LIN {X 0,Y 315.719,Z 733.66,A -85,B 0,C 180,E1 14074.745,E2 14074.745} C_VEL
LIN {X 0,Y 317.887,Z 739.054,A -85,B 0,C 180,E1 14075.526,E2 14075.526} C_VEL
LIN {X 0,Y 320.748,Z 743.078,A -85,B 0,C 180,E1 14076.392,E2 14076.392} C_VEL
LIN {X 0,Y 337.492,Z 768.828,A -85,B 0,C 180,E1 14081.01,E2 14081.01} C_VEL
LIN {X 0,Y 351.27,Z 797.337,A -85,B 0,C 180,E1 14085.073,E2 14085.073} C_VEL
LIN {X 0,Y 359.237,Z 823.028,A -85,B 0,C 180,E1 14088.326,E2 14088.326} C_VEL
LIN {X 0,Y 352.116,Z 857.888,A -85,B 0,C 180,E1 14091.071,E2 14091.071} C_VEL
LIN {X 0,Y 344.17,Z 888.383,A -85,B 0,C 180,E1 14094.581,E2 14094.581} C_VEL
LIN {X 0,Y 336.227,Z 914.82,A -85,B 0,C 180,E1 14098.833,E2 14098.833} C_VEL
LIN {X 0,Y 328.748,Z 938.426,A -85,B 0,C 180,E1 14104.142,E2 14104.142} C_VEL
LIN {X 0,Y 323.256,Z 956.658,A -85,B 0,C 180,E1 14110.032,E2 14110.032} C_VEL
LIN {X 0,Y 319.91,Z 969.689,A -85,B 0,C 180,E1 14116.312,E2 14116.312} C_VEL
LIN {X 0,Y 318.308,Z 977.967,A -85,B 0,C 180,E1 14123.171,E2 14123.171} C_VEL
LIN {X 0,Y 318.122,Z 980.655,A -85,B 0,C 180,E1 14130,E2 14130} C_VEL
LIN {X 0,Y 318.325,Z 977.878,A -85,B 0,C 180,E1 14136.83,E2 14136.83} C_VEL
LIN {X 0,Y 319.962,Z 969.528,A -85,B 0,C 180,E1 14143.687,E2 14143.687} C_VEL
LIN {X 0,Y 323.345,Z 956.356,A -85,B 0,C 180,E1 14149.986,E2 14149.986} C_VEL
LIN {X 0,Y 328.917,Z 937.87,A -85,B 0,C 180,E1 14155.897,E2 14155.897} C_VEL
LIN {X 0,Y 336.458,Z 913.934,A -85,B 0,C 180,E1 14161.232,E2 14161.232} C_VEL
LIN {X 0,Y 344.929,Z 885.442,A -85,B 0,C 180,E1 14165.728,E2 14165.728} C_VEL
LIN {X 0,Y 353.166,Z 852.828,A -85,B 0,C 180,E1 14169.299,E2 14169.299} C_VEL
LIN {X 0,Y 359.003,Z 821.032,A -85,B 0,C 180,E1 14171.77,E2 14171.77} C_VEL
LIN {X 0,Y 348.714,Z 791.49,A -85,B 0,C 180,E1 14175.622,E2 14175.622} C_VEL
LIN {X 0,Y 333.855,Z 762.92,A -85,B 0,C 180,E1 14179.841,E2 14179.841} C_VEL
LIN {X 0,Y 318.479,Z 739.646,A -85,B 0,C 180,E1 14184.163,E2 14184.163} C_VEL
LIN {X 0,Y 315.762,Z 734.408,A -85,B 0,C 180,E1 14185.064,E2 14185.064} C_VEL
LIN {X 0,Y 315.891,Z 733.66,A -85,B 0,C 180,E1 14191.354,E2 14191.354} C_VEL
LIN {X 0,Y 316.196,Z 733.66,A -85,B 0,C 180,E1 14197.47,E2 14197.47} C_VEL
LIN {X 0,Y 316.495,Z 733.66,A -85,B 0,C 180,E1 14203.314,E2 14203.314} C_VEL
LIN {X 0,Y 317.022,Z 733.66,A -85,B 0,C 180,E1 14211.757,E2 14211.757} C_VEL
LIN {X 0,Y 317.696,Z 733.66,A -85,B 0,C 180,E1 14219.994,E2 14219.994} C_VEL
LIN {X 0,Y 317.039,Z 733.66,A -85,B 0,C 180,E1 14228.231,E2 14228.231} C_VEL
LIN {X 0,Y 316.543,Z 733.66,A -85,B 0,C 180,E1 14236.671,E2 14236.671} C_VEL
LIN {X 0,Y 316.1,Z 733.66,A -85,B 0,C 180,E1 14244.482,E2 14244.482} C_VEL
LIN {X 0,Y 315.775,Z 733.66,A -85,B 0,C 180,E1 14251.823,E2 14251.823} C_VEL
LIN {X 0,Y 315.754,Z 733.66,A -85,B 0,C 180,E1 14254.342,E2 14254.342} C_VEL
LIN {X 0,Y 317.927,Z 739.136,A -85,B 0,C 180,E1 14255.152,E2 14255.152} C_VEL
LIN {X 0,Y 321.023,Z 743.491,A -85,B 0,C 180,E1 14256.083,E2 14256.083} C_VEL
LIN {X 0,Y 336.553,Z 767.239,A -85,B 0,C 180,E1 14260.305,E2 14260.305} C_VEL
LIN {X 0,Y 350.017,Z 791.741,A -85,B 0,C 180,E1 14263.573,E2 14263.573} C_VEL
LIN {X 0,Y 360.355,Z 827.54,A -85,B 0,C 180,E1 14267.003,E2 14267.003} C_VEL
LIN {X 0,Y 354.186,Z 864.729,A -85,B 0,C 180,E1 14269.179,E2 14269.179} C_VEL
LIN {X 0,Y 346.202,Z 898.964,A -85,B 0,C 180,E1 14272.245,E2 14272.245} C_VEL
LIN {X 0,Y 337.789,Z 929.303,A -85,B 0,C 180,E1 14276.16,E2 14276.16} C_VEL
LIN {X 0,Y 329.891,Z 956.501,A -85,B 0,C 180,E1 14281.15,E2 14281.15} C_VEL
LIN {X 0,Y 323.714,Z 978.764,A -85,B 0,C 180,E1 14286.938,E2 14286.938} C_VEL
LIN {X 0,Y 319.815,Z 996.193,A -85,B 0,C 180,E1 14293.497,E2 14293.497} C_VEL
LIN {X 0,Y 318.446,Z 1005.836,A -85,B 0,C 180,E1 14299.036,E2 14299.036} C_VEL
LIN {X 0,Y 318.166,Z 1011.498,A -85,B 0,C 180,E1 14304.538,E2 14304.538} C_VEL
LIN {X 0,Y 318.196,Z 1013.428,A -85,B 0,C 180,E1 14310,E2 14310} C_VEL
LIN {X 0,Y 318.188,Z 1011.507,A -85,B 0,C 180,E1 14315.461,E2 14315.461} C_VEL
LIN {X 0,Y 318.486,Z 1005.851,A -85,B 0,C 180,E1 14320.962,E2 14320.962} C_VEL
LIN {X 0,Y 320.15,Z 994.65,A -85,B 0,C 180,E1 14327.192,E2 14327.192} C_VEL
LIN {X 0,Y 324.095,Z 977.701,A -85,B 0,C 180,E1 14333.397,E2 14333.397} C_VEL
LIN {X 0,Y 330.329,Z 955.266,A -85,B 0,C 180,E1 14339.134,E2 14339.134} C_VEL
LIN {X 0,Y 338.372,Z 927.731,A -85,B 0,C 180,E1 14344.078,E2 14344.078} C_VEL
LIN {X 0,Y 344.691,Z 905.27,A -85,B 0,C 180,E1 14347.058,E2 14347.058} C_VEL
LIN {X 0,Y 345.028,Z 891.788,A -85,B 0,C 180,E1 14348.915,E2 14348.915} C_VEL
LIN {X 0,Y 344.878,Z 879.547,A -85,B 0,C 180,E1 14350.45,E2 14350.45} C_VEL
LIN {X 0,Y 345.262,Z 877.652,A -85,B 0,C 180,E1 14350.624,E2 14350.624} C_VEL
LIN {X 0,Y 352.782,Z 841.115,A -85,B 0,C 180,E1 14353.157,E2 14353.157} C_VEL
LIN {X 0,Y 354.632,Z 826.28,A -85,B 0,C 180,E1 14353.945,E2 14353.945} C_VEL
LIN {X 0,Y 353.828,Z 815.884,A -85,B 0,C 180,E1 14354.939,E2 14354.939} C_VEL
LIN {X 0,Y 354.413,Z 805.731,A -85,B 0,C 180,E1 14356.89,E2 14356.89} C_VEL
LIN {X 0,Y 352.564,Z 801.602,A -85,B 0,C 180,E1 14359.906,E2 14359.906} C_VEL
LIN {X 0,Y 352.295,Z 802.737,A -85,B 0,C 180,E1 14363.018,E2 14363.018} C_VEL
LIN {X 0,Y 352.883,Z 809.058,A -85,B 0,C 180,E1 14365.545,E2 14365.545} C_VEL
LIN {X 0,Y 343.129,Z 843.636,A -85,B 0,C 180,E1 14368.963,E2 14368.963} C_VEL
LIN {X 0,Y 335.37,Z 867.34,A -85,B 0,C 180,E1 14372.482,E2 14372.482} C_VEL
LIN {X 0,Y 327.758,Z 887.089,A -85,B 0,C 180,E1 14376.888,E2 14376.888} C_VEL
LIN {X 0,Y 321.86,Z 900.268,A -85,B 0,C 180,E1 14381.494,E2 14381.494} C_VEL
LIN {X 0,Y 317.622,Z 908.248,A -85,B 0,C 180,E1 14386.218,E2 14386.218} C_VEL
LIN {X 0,Y 314.61,Z 911.796,A -85,B 0,C 180,E1 14391.705,E2 14391.705} C_VEL
LIN {X 0,Y 313.23,Z 909.746,A -85,B 0,C 180,E1 14397.236,E2 14397.236} C_VEL
LIN {X 0,Y 313.169,Z 901.828,A -85,B 0,C 180,E1 14402.777,E2 14402.777} C_VEL
LIN {X 0,Y 314.276,Z 888.435,A -85,B 0,C 180,E1 14407.967,E2 14407.967} C_VEL
LIN {X 0,Y 316.237,Z 870.789,A -85,B 0,C 180,E1 14412.448,E2 14412.448} C_VEL
LIN {X 0,Y 319.015,Z 847.121,A -85,B 0,C 180,E1 14416.55,E2 14416.55} C_VEL
LIN {X 0,Y 321.875,Z 820.749,A -85,B 0,C 180,E1 14419.65,E2 14419.65} C_VEL
LIN {X 0,Y 324.187,Z 789.991,A -85,B 0,C 180,E1 14421.945,E2 14421.945} C_VEL
LIN {X 0,Y 310.002,Z 740.414,A -85,B 0,C 180,E1 14425.18,E2 14425.18} C_VEL
LIN {X 0,Y 308.125,Z 733.66,A -85,B 0,C 180,E1 14425.647,E2 14425.647} C_VEL
LIN {X 0,Y 307.834,Z 733.76,A -85,B 0,C 180,E1 14432.566,E2 14432.566} C_VEL
LIN {X 0,Y 310.075,Z 739.153,A -85,B 0,C 180,E1 14433.438,E2 14433.438} C_VEL
LIN {X 0,Y 312.739,Z 742.517,A -85,B 0,C 180,E1 14434.311,E2 14434.311} C_VEL
LIN {X 0,Y 328.649,Z 766.861,A -85,B 0,C 180,E1 14439.098,E2 14439.098} C_VEL
LIN {X 0,Y 342.598,Z 793.742,A -85,B 0,C 180,E1 14443.318,E2 14443.318} C_VEL
LIN {X 0,Y 352.285,Z 821.897,A -85,B 0,C 180,E1 14447.171,E2 14447.171} C_VEL
LIN {X 0,Y 352.391,Z 828.572,A -85,B 0,C 180,E1 14447.809,E2 14447.809} C_VEL
LIN {X 0,Y 344.891,Z 862.553,A -85,B 0,C 180,E1 14450.676,E2 14450.676} C_VEL
LIN {X 0,Y 336.417,Z 893.037,A -85,B 0,C 180,E1 14454.39,E2 14454.39} C_VEL
LIN {X 0,Y 327.713,Z 920.477,A -85,B 0,C 180,E1 14459.161,E2 14459.161} C_VEL
LIN {X 0,Y 320.127,Z 943.273,A -85,B 0,C 180,E1 14464.807,E2 14464.807} C_VEL
LIN {X 0,Y 314.687,Z 960.699,A -85,B 0,C 180,E1 14471.049,E2 14471.049} C_VEL
LIN {X 0,Y 311.683,Z 972.269,A -85,B 0,C 180,E1 14477.374,E2 14477.374} C_VEL
LIN {X 0,Y 310.313,Z 979.325,A -85,B 0,C 180,E1 14484.4,E2 14484.4} C_VEL
LIN {X 0,Y 310.245,Z 981.06,A -85,B 0,C 180,E1 14490,E2 14490} C_VEL
LIN {X 0,Y 310.473,Z 978.285,A -85,B 0,C 180,E1 14497.003,E2 14497.003} C_VEL
LIN {X 0,Y 312.248,Z 969.827,A -85,B 0,C 180,E1 14504.104,E2 14504.104} C_VEL
LIN {X 0,Y 316.145,Z 955.711,A -85,B 0,C 180,E1 14510.9,E2 14510.9} C_VEL
LIN {X 0,Y 322.48,Z 935.952,A -85,B 0,C 180,E1 14517.134,E2 14517.134} C_VEL
LIN {X 0,Y 330.754,Z 911.07,A -85,B 0,C 180,E1 14522.574,E2 14522.574} C_VEL
LIN {X 0,Y 339.489,Z 882.48,A -85,B 0,C 180,E1 14526.939,E2 14526.939} C_VEL
LIN {X 0,Y 347.64,Z 850.852,A -85,B 0,C 180,E1 14530.339,E2 14530.339} C_VEL
LIN {X 0,Y 352.866,Z 824.113,A -85,B 0,C 180,E1 14532.427,E2 14532.427} C_VEL
LIN {X 0,Y 342.854,Z 794.622,A -85,B 0,C 180,E1 14536.463,E2 14536.463} C_VEL
LIN {X 0,Y 328.84,Z 767.242,A -85,B 0,C 180,E1 14540.716,E2 14540.716} C_VEL
LIN {X 0,Y 314.245,Z 745.05,A -85,B 0,C 180,E1 14545.044,E2 14545.044} C_VEL
LIN {X 0,Y 310.585,Z 739.636,A -85,B 0,C 180,E1 14546.254,E2 14546.254} C_VEL
LIN {X 0,Y 307.873,Z 734.455,A -85,B 0,C 180,E1 14547.245,E2 14547.245} C_VEL
LIN {X 0,Y 308.049,Z 733.66,A -85,B 0,C 180,E1 14553.74,E2 14553.74} C_VEL
LIN {X 0,Y 308.391,Z 733.66,A -85,B 0,C 180,E1 14559.893,E2 14559.893} C_VEL
LIN {X 0,Y 308.644,Z 733.66,A -85,B 0,C 180,E1 14565.796,E2 14565.796} C_VEL
LIN {X 0,Y 309.312,Z 733.66,A -85,B 0,C 180,E1 14574.376,E2 14574.376} C_VEL
LIN {X 0,Y 309.792,Z 733.66,A -85,B 0,C 180,E1 14579.994,E2 14579.994} C_VEL
LIN {X 0,Y 309.097,Z 733.66,A -85,B 0,C 180,E1 14588.444,E2 14588.444} C_VEL
LIN {X 0,Y 308.596,Z 733.66,A -85,B 0,C 180,E1 14597.113,E2 14597.113} C_VEL
LIN {X 0,Y 308.217,Z 733.66,A -85,B 0,C 180,E1 14603.133,E2 14603.133} C_VEL
LIN {X 0,Y 307.864,Z 733.66,A -85,B 0,C 180,E1 14611.215,E2 14611.215} C_VEL
LIN {X 0,Y 307.871,Z 733.66,A -85,B 0,C 180,E1 14612.165,E2 14612.165} C_VEL
LIN {X 0,Y 310.1,Z 739.211,A -85,B 0,C 180,E1 14613.067,E2 14613.067} C_VEL
LIN {X 0,Y 312.757,Z 742.554,A -85,B 0,C 180,E1 14613.934,E2 14613.934} C_VEL
LIN {X 0,Y 329.952,Z 768.564,A -85,B 0,C 180,E1 14618.991,E2 14618.991} C_VEL
LIN {X 0,Y 344.988,Z 795.969,A -85,B 0,C 180,E1 14622.854,E2 14622.854} C_VEL
LIN {X 0,Y 354.429,Z 830.867,A -85,B 0,C 180,E1 14626.343,E2 14626.343} C_VEL
LIN {X 0,Y 347.762,Z 866.235,A -85,B 0,C 180,E1 14628.466,E2 14628.466} C_VEL
LIN {X 0,Y 339.854,Z 898.559,A -85,B 0,C 180,E1 14631.411,E2 14631.411} C_VEL
LIN {X 0,Y 331.048,Z 929.012,A -85,B 0,C 180,E1 14635.397,E2 14635.397} C_VEL
LIN {X 0,Y 322.614,Z 956.671,A -85,B 0,C 180,E1 14640.588,E2 14640.588} C_VEL
LIN {X 0,Y 316.476,Z 977.674,A -85,B 0,C 180,E1 14646.151,E2 14646.151} C_VEL
LIN {X 0,Y 312.377,Z 994.208,A -85,B 0,C 180,E1 14652.365,E2 14652.365} C_VEL
LIN {X 0,Y 310.585,Z 1005.423,A -85,B 0,C 180,E1 14658.755,E2 14658.755} C_VEL
LIN {X 0,Y 310.267,Z 1011.089,A -85,B 0,C 180,E1 14664.399,E2 14664.399} C_VEL
LIN {X 0,Y 310.314,Z 1013.022,A -85,B 0,C 180,E1 14670,E2 14670} C_VEL
LIN {X 0,Y 310.288,Z 1011.099,A -85,B 0,C 180,E1 14675.6,E2 14675.6} C_VEL
LIN {X 0,Y 310.832,Z 1004.069,A -85,B 0,C 180,E1 14682.218,E2 14682.218} C_VEL
LIN {X 0,Y 313.101,Z 991.048,A -85,B 0,C 180,E1 14689.051,E2 14689.051} C_VEL
LIN {X 0,Y 317.903,Z 972.612,A -85,B 0,C 180,E1 14695.381,E2 14695.381} C_VEL
LIN {X 0,Y 324.742,Z 949.962,A -85,B 0,C 180,E1 14700.855,E2 14700.855} C_VEL
LIN {X 0,Y 333.393,Z 921.91,A -85,B 0,C 180,E1 14705.671,E2 14705.671} C_VEL
LIN {X 0,Y 342.039,Z 890.249,A -85,B 0,C 180,E1 14709.475,E2 14709.475} C_VEL
LIN {X 0,Y 345.262,Z 877.652,A -85,B 0,C 180,E1 14710.624,E2 14710.624} C_VEL
LIN {X 0,Y 345.636,Z 862.952,A -85,B 0,C 180,E1 14712.213,E2 14712.213} C_VEL
LIN {X 0,Y 345.686,Z 847.734,A -85,B 0,C 180,E1 14713.652,E2 14713.652} C_VEL
LIN {X 0,Y 348.589,Z 827.915,A -85,B 0,C 180,E1 14714.778,E2 14714.778} C_VEL
LIN {X 0,Y 349.864,Z 816.657,A -85,B 0,C 180,E1 14716.342,E2 14716.342} C_VEL
LIN {X 0,Y 350.407,Z 812.2,A -85,B 0,C 180,E1 14717.27,E2 14717.27} C_VEL
LIN {X 0,Y 349.152,Z 809.136,A -85,B 0,C 180,E1 14719.433,E2 14719.433} C_VEL
LIN {X 0,Y 348.638,Z 809.515,A -85,B 0,C 180,E1 14722.564,E2 14722.564} C_VEL
LIN {X 0,Y 348.845,Z 813.277,A -85,B 0,C 180,E1 14724.507,E2 14724.507} C_VEL
LIN {X 0,Y 336.466,Z 851.174,A -85,B 0,C 180,E1 14728.657,E2 14728.657} C_VEL
LIN {X 0,Y 327.878,Z 874.081,A -85,B 0,C 180,E1 14732.506,E2 14732.506} C_VEL
LIN {X 0,Y 319.961,Z 892.066,A -85,B 0,C 180,E1 14737.029,E2 14737.029} C_VEL
LIN {X 0,Y 313.274,Z 905.19,A -85,B 0,C 180,E1 14742.426,E2 14742.426} C_VEL
LIN {X 0,Y 309.131,Z 911.475,A -85,B 0,C 180,E1 14747.274,E2 14747.274} C_VEL
LIN {X 0,Y 306.931,Z 913.336,A -85,B 0,C 180,E1 14751.496,E2 14751.496} C_VEL
LIN {X 0,Y 305.425,Z 910.977,A -85,B 0,C 180,E1 14757.165,E2 14757.165} C_VEL
LIN {X 0,Y 305.353,Z 902.819,A -85,B 0,C 180,E1 14762.848,E2 14762.848} C_VEL
LIN {X 0,Y 306.49,Z 889.121,A -85,B 0,C 180,E1 14768.171,E2 14768.171} C_VEL
LIN {X 0,Y 308.771,Z 869.532,A -85,B 0,C 180,E1 14773.114,E2 14773.114} C_VEL
LIN {X 0,Y 311.579,Z 846.035,A -85,B 0,C 180,E1 14777.139,E2 14777.139} C_VEL
LIN {X 0,Y 314.582,Z 818.438,A -85,B 0,C 180,E1 14780.308,E2 14780.308} C_VEL
LIN {X 0,Y 316.404,Z 789.468,A -85,B 0,C 180,E1 14782.459,E2 14782.459} C_VEL
LIN {X 0,Y 300.116,Z 733.66,A -85,B 0,C 180,E1 14786.454,E2 14786.454} C_VEL
LIN {X 0,Y 299.966,Z 733.66,A -85,B 0,C 180,E1 14790.097,E2 14790.097} C_VEL
LIN {X 0,Y 301.982,Z 738.935,A -85,B 0,C 180,E1 14791.005,E2 14791.005} C_VEL
LIN {X 0,Y 305.006,Z 742.493,A -85,B 0,C 180,E1 14792.101,E2 14792.101} C_VEL
LIN {X 0,Y 320.547,Z 765.584,A -85,B 0,C 180,E1 14797.201,E2 14797.201} C_VEL
LIN {X 0,Y 334.503,Z 791.877,A -85,B 0,C 180,E1 14801.673,E2 14801.673} C_VEL
LIN {X 0,Y 344.06,Z 817.214,A -85,B 0,C 180,E1 14805.397,E2 14805.397} C_VEL
LIN {X 0,Y 346.837,Z 827.807,A -85,B 0,C 180,E1 14806.856,E2 14806.856} C_VEL
LIN {X 0,Y 338.826,Z 862.802,A -85,B 0,C 180,E1 14809.812,E2 14809.812} C_VEL
LIN {X 0,Y 330.004,Z 893.431,A -85,B 0,C 180,E1 14813.589,E2 14813.589} C_VEL
LIN {X 0,Y 320.835,Z 920.937,A -85,B 0,C 180,E1 14818.439,E2 14818.439} C_VEL
LIN {X 0,Y 312.87,Z 943.681,A -85,B 0,C 180,E1 14824.181,E2 14824.181} C_VEL
LIN {X 0,Y 307.124,Z 961.108,A -85,B 0,C 180,E1 14830.564,E2 14830.564} C_VEL
LIN {X 0,Y 303.876,Z 972.875,A -85,B 0,C 180,E1 14837.201,E2 14837.201} C_VEL
LIN {X 0,Y 302.441,Z 979.732,A -85,B 0,C 180,E1 14844.254,E2 14844.254} C_VEL
LIN {X 0,Y 302.37,Z 981.466,A -85,B 0,C 180,E1 14850,E2 14850} C_VEL
LIN {X 0,Y 302.609,Z 978.694,A -85,B 0,C 180,E1 14857.186,E2 14857.186} C_VEL
LIN {X 0,Y 304.494,Z 970.35,A -85,B 0,C 180,E1 14864.397,E2 14864.397} C_VEL
LIN {X 0,Y 308.649,Z 956.253,A -85,B 0,C 180,E1 14871.381,E2 14871.381} C_VEL
LIN {X 0,Y 315.139,Z 937.036,A -85,B 0,C 180,E1 14877.617,E2 14877.617} C_VEL
LIN {X 0,Y 323.286,Z 913.635,A -85,B 0,C 180,E1 14882.919,E2 14882.919} C_VEL
LIN {X 0,Y 332.374,Z 885.51,A -85,B 0,C 180,E1 14887.428,E2 14887.428} C_VEL
LIN {X 0,Y 341.118,Z 853.362,A -85,B 0,C 180,E1 14891.008,E2 14891.008} C_VEL
LIN {X 0,Y 346.7,Z 826.973,A -85,B 0,C 180,E1 14893.137,E2 14893.137} C_VEL
LIN {X 0,Y 336.73,Z 796.898,A -85,B 0,C 180,E1 14897.434,E2 14897.434} C_VEL
LIN {X 0,Y 322.725,Z 769.328,A -85,B 0,C 180,E1 14901.987,E2 14901.987} C_VEL
LIN {X 0,Y 307.57,Z 746.275,A -85,B 0,C 180,E1 14906.832,E2 14906.832} C_VEL
LIN {X 0,Y 302.999,Z 739.88,A -85,B 0,C 180,E1 14908.478,E2 14908.478} C_VEL
LIN {X 0,Y 300.168,Z 735.451,A -85,B 0,C 180,E1 14909.587,E2 14909.587} C_VEL
LIN {X 0,Y 299.981,Z 733.66,A -85,B 0,C 180,E1 14909.904,E2 14909.904} C_VEL
LIN {X 0,Y 300.215,Z 733.66,A -85,B 0,C 180,E1 14916.199,E2 14916.199} C_VEL
LIN {X 0,Y 300.662,Z 733.66,A -85,B 0,C 180,E1 14923.102,E2 14923.102} C_VEL
LIN {X 0,Y 301.125,Z 733.66,A -85,B 0,C 180,E1 14931.746,E2 14931.746} C_VEL
LIN {X 0,Y 301.899,Z 733.66,A -85,B 0,C 180,E1 14939.994,E2 14939.994} C_VEL
LIN {X 0,Y 301.42,Z 733.66,A -85,B 0,C 180,E1 14945.759,E2 14945.759} C_VEL
LIN {X 0,Y 301.006,Z 733.66,A -85,B 0,C 180,E1 14951.6,E2 14951.6} C_VEL
LIN {X 0,Y 300.605,Z 733.66,A -85,B 0,C 180,E1 14957.582,E2 14957.582} C_VEL
LIN {X 0,Y 300.128,Z 733.66,A -85,B 0,C 180,E1 14964.759,E2 14964.759} C_VEL
LIN {X 0,Y 299.989,Z 733.777,A -85,B 0,C 180,E1 14969.751,E2 14969.751} C_VEL
LIN {X 0,Y 302.001,Z 738.972,A -85,B 0,C 180,E1 14970.641,E2 14970.641} C_VEL
LIN {X 0,Y 305.02,Z 742.516,A -85,B 0,C 180,E1 14971.73,E2 14971.73} C_VEL
LIN {X 0,Y 320.804,Z 765.937,A -85,B 0,C 180,E1 14976.852,E2 14976.852} C_VEL
LIN {X 0,Y 338.185,Z 796.442,A -85,B 0,C 180,E1 14981.639,E2 14981.639} C_VEL
LIN {X 0,Y 346.476,Z 824.437,A -85,B 0,C 180,E1 14984.675,E2 14984.675} C_VEL
LIN {X 0,Y 347.971,Z 834.858,A -85,B 0,C 180,E1 14985.66,E2 14985.66} C_VEL
LIN {X 0,Y 340.883,Z 869.798,A -85,B 0,C 180,E1 14987.881,E2 14987.881} C_VEL
LIN {X 0,Y 332.061,Z 903.71,A -85,B 0,C 180,E1 14991.174,E2 14991.174} C_VEL
LIN {X 0,Y 322.769,Z 933.948,A -85,B 0,C 180,E1 14995.474,E2 14995.474} C_VEL
LIN {X 0,Y 314.344,Z 960.057,A -85,B 0,C 180,E1 15000.754,E2 15000.754} C_VEL
LIN {X 0,Y 307.866,Z 981.184,A -85,B 0,C 180,E1 15006.831,E2 15006.831} C_VEL
LIN {X 0,Y 304.069,Z 996.753,A -85,B 0,C 180,E1 15013.362,E2 15013.362} C_VEL
LIN {X 0,Y 302.577,Z 1006.786,A -85,B 0,C 180,E1 15019.913,E2 15019.913} C_VEL
LIN {X 0,Y 302.383,Z 1010.681,A -85,B 0,C 180,E1 15024.252,E2 15024.252} C_VEL
LIN {X 0,Y 302.422,Z 1012.615,A -85,B 0,C 180,E1 15030,E2 15030} C_VEL
LIN {X 0,Y 302.402,Z 1010.691,A -85,B 0,C 180,E1 15035.747,E2 15035.747} C_VEL
LIN {X 0,Y 302.964,Z 1003.837,A -85,B 0,C 180,E1 15042.408,E2 15042.408} C_VEL
LIN {X 0,Y 305.238,Z 991.599,A -85,B 0,C 180,E1 15049.119,E2 15049.119} C_VEL
LIN {X 0,Y 310.107,Z 973.861,A -85,B 0,C 180,E1 15055.54,E2 15055.54} C_VEL
LIN {X 0,Y 317.27,Z 951.185,A -85,B 0,C 180,E1 15061.261,E2 15061.261} C_VEL
LIN {X 0,Y 326.232,Z 923.463,A -85,B 0,C 180,E1 15066.202,E2 15066.202} C_VEL
LIN {X 0,Y 335.554,Z 891.084,A -85,B 0,C 180,E1 15070.224,E2 15070.224} C_VEL
LIN {X 0,Y 343.855,Z 856.887,A -85,B 0,C 180,E1 15073.069,E2 15073.069} C_VEL
LIN {X 0,Y 345.686,Z 847.734,A -85,B 0,C 180,E1 15073.652,E2 15073.652} C_VEL
LIN {X 0,Y 346.221,Z 836.168,A -85,B 0,C 180,E1 15074.708,E2 15074.708} C_VEL
LIN {X 0,Y 345.537,Z 823.234,A -85,B 0,C 180,E1 15076.758,E2 15076.758} C_VEL
LIN {X 0,Y 345.882,Z 820.398,A -85,B 0,C 180,E1 15077.334,E2 15077.334} C_VEL
LIN {X 0,Y 346.161,Z 817.854,A -85,B 0,C 180,E1 15078.036,E2 15078.036} C_VEL
LIN {X 0,Y 344.974,Z 815.915,A -85,B 0,C 180,E1 15080.961,E2 15080.961} C_VEL
LIN {X 0,Y 345.027,Z 818.601,A -85,B 0,C 180,E1 15083.703,E2 15083.703} C_VEL
LIN {X 0,Y 332.022,Z 852.806,A -85,B 0,C 180,E1 15087.547,E2 15087.547} C_VEL
LIN {X 0,Y 322.681,Z 875.238,A -85,B 0,C 180,E1 15091.385,E2 15091.385} C_VEL
LIN {X 0,Y 313.697,Z 893.828,A -85,B 0,C 180,E1 15096.165,E2 15096.165} C_VEL
LIN {X 0,Y 306.779,Z 906.153,A -85,B 0,C 180,E1 15101.296,E2 15101.296} C_VEL
LIN {X 0,Y 301.623,Z 913.274,A -85,B 0,C 180,E1 15106.952,E2 15106.952} C_VEL
LIN {X 0,Y 299.259,Z 914.884,A -85,B 0,C 180,E1 15111.277,E2 15111.277} C_VEL
LIN {X 0,Y 297.62,Z 912.2,A -85,B 0,C 180,E1 15117.091,E2 15117.091} C_VEL
LIN {X 0,Y 297.544,Z 903.759,A -85,B 0,C 180,E1 15122.923,E2 15122.923} C_VEL
LIN {X 0,Y 298.718,Z 889.791,A -85,B 0,C 180,E1 15128.385,E2 15128.385} C_VEL
LIN {X 0,Y 300.836,Z 871.565,A -85,B 0,C 180,E1 15133.096,E2 15133.096} C_VEL
LIN {X 0,Y 303.856,Z 847.188,A -85,B 0,C 180,E1 15137.402,E2 15137.402} C_VEL
LIN {X 0,Y 307.022,Z 819.196,A -85,B 0,C 180,E1 15140.705,E2 15140.705} C_VEL
LIN {X 0,Y 308.909,Z 791.09,A -85,B 0,C 180,E1 15142.847,E2 15142.847} C_VEL
LIN {X 0,Y 292.956,Z 736.992,A -85,B 0,C 180,E1 15146.706,E2 15146.706} C_VEL
LIN {X 0,Y 292.199,Z 733.66,A -85,B 0,C 180,E1 15147.002,E2 15147.002} C_VEL
LIN {X 0,Y 292.299,Z 735.133,A -85,B 0,C 180,E1 15147.453,E2 15147.453} C_VEL
LIN {X 0,Y 295.312,Z 740.026,A -85,B 0,C 180,E1 15148.812,E2 15148.812} C_VEL
LIN {X 0,Y 297.348,Z 742.62,A -85,B 0,C 180,E1 15149.65,E2 15149.65} C_VEL
LIN {X 0,Y 310.753,Z 762.087,A -85,B 0,C 180,E1 15154.563,E2 15154.563} C_VEL
LIN {X 0,Y 325.311,Z 787.42,A -85,B 0,C 180,E1 15159.47,E2 15159.47} C_VEL
LIN {X 0,Y 336.392,Z 814.875,A -85,B 0,C 180,E1 15163.839,E2 15163.839} C_VEL
LIN {X 0,Y 340.31,Z 831.716,A -85,B 0,C 180,E1 15166.192,E2 15166.192} C_VEL
LIN {X 0,Y 331.988,Z 866.244,A -85,B 0,C 180,E1 15169.248,E2 15169.248} C_VEL
LIN {X 0,Y 322.484,Z 897.231,A -85,B 0,C 180,E1 15173.272,E2 15173.272} C_VEL
LIN {X 0,Y 313.625,Z 922.475,A -85,B 0,C 180,E1 15177.924,E2 15177.924} C_VEL
LIN {X 0,Y 305.268,Z 945.257,A -85,B 0,C 180,E1 15183.884,E2 15183.884} C_VEL
LIN {X 0,Y 299.106,Z 963.018,A -85,B 0,C 180,E1 15190.79,E2 15190.79} C_VEL
LIN {X 0,Y 296.02,Z 973.638,A -85,B 0,C 180,E1 15197.143,E2 15197.143} C_VEL
LIN {X 0,Y 294.564,Z 980.139,A -85,B 0,C 180,E1 15204.1,E2 15204.1} C_VEL
LIN {X 0,Y 294.478,Z 981.872,A -85,B 0,C 180,E1 15210,E2 15210} C_VEL
LIN {X 0,Y 294.763,Z 979.102,A -85,B 0,C 180,E1 15217.379,E2 15217.379} C_VEL
LIN {X 0,Y 296.784,Z 970.76,A -85,B 0,C 180,E1 15224.779,E2 15224.779} C_VEL
LIN {X 0,Y 300.987,Z 957.283,A -85,B 0,C 180,E1 15231.685,E2 15231.685} C_VEL
LIN {X 0,Y 307.887,Z 937.925,A -85,B 0,C 180,E1 15238.177,E2 15238.177} C_VEL
LIN {X 0,Y 316.467,Z 914.472,A -85,B 0,C 180,E1 15243.618,E2 15243.618} C_VEL
LIN {X 0,Y 326.308,Z 885.259,A -85,B 0,C 180,E1 15248.36,E2 15248.36} C_VEL
LIN {X 0,Y 335.483,Z 852.598,A -85,B 0,C 180,E1 15252.001,E2 15252.001} C_VEL
LIN {X 0,Y 340.635,Z 830.346,A -85,B 0,C 180,E1 15253.783,E2 15253.783} C_VEL
LIN {X 0,Y 331.622,Z 801.801,A -85,B 0,C 180,E1 15258.048,E2 15258.048} C_VEL
LIN {X 0,Y 318.815,Z 775.237,A -85,B 0,C 180,E1 15262.622,E2 15262.622} C_VEL
LIN {X 0,Y 304.276,Z 752.583,A -85,B 0,C 180,E1 15267.528,E2 15267.528} C_VEL
LIN {X 0,Y 295.763,Z 740.318,A -85,B 0,C 180,E1 15270.849,E2 15270.849} C_VEL
LIN {X 0,Y 292.323,Z 735.34,A -85,B 0,C 180,E1 15272.355,E2 15272.355} C_VEL
LIN {X 0,Y 292.182,Z 733.66,A -85,B 0,C 180,E1 15272.779,E2 15272.779} C_VEL
LIN {X 0,Y 292.432,Z 733.66,A -85,B 0,C 180,E1 15278.745,E2 15278.745} C_VEL
LIN {X 0,Y 292.774,Z 733.66,A -85,B 0,C 180,E1 15285.008,E2 15285.008} C_VEL
LIN {X 0,Y 293.174,Z 733.66,A -85,B 0,C 180,E1 15291.75,E2 15291.75} C_VEL
LIN {X 0,Y 293.994,Z 733.66,A -85,B 0,C 180,E1 15299.993,E2 15299.993} C_VEL
LIN {X 0,Y 293.482,Z 733.66,A -85,B 0,C 180,E1 15305.915,E2 15305.915} C_VEL
LIN {X 0,Y 293.051,Z 733.66,A -85,B 0,C 180,E1 15311.92,E2 15311.92} C_VEL
LIN {X 0,Y 292.615,Z 733.66,A -85,B 0,C 180,E1 15318.079,E2 15318.079} C_VEL
LIN {X 0,Y 292.198,Z 733.775,A -85,B 0,C 180,E1 15326.989,E2 15326.989} C_VEL
LIN {X 0,Y 293.959,Z 738.742,A -85,B 0,C 180,E1 15327.901,E2 15327.901} C_VEL
LIN {X 0,Y 297.302,Z 742.5,A -85,B 0,C 180,E1 15329.262,E2 15329.262} C_VEL
LIN {X 0,Y 311.292,Z 763.009,A -85,B 0,C 180,E1 15334.356,E2 15334.356} C_VEL
LIN {X 0,Y 326.553,Z 787.892,A -85,B 0,C 180,E1 15338.954,E2 15338.954} C_VEL
LIN {X 0,Y 335.82,Z 807.992,A -85,B 0,C 180,E1 15341.782,E2 15341.782} C_VEL
LIN {X 0,Y 342.137,Z 835.631,A -85,B 0,C 180,E1 15344.79,E2 15344.79} C_VEL
LIN {X 0,Y 334.945,Z 869.686,A -85,B 0,C 180,E1 15346.989,E2 15346.989} C_VEL
LIN {X 0,Y 325.631,Z 903.946,A -85,B 0,C 180,E1 15350.366,E2 15350.366} C_VEL
LIN {X 0,Y 316.19,Z 933.32,A -85,B 0,C 180,E1 15354.603,E2 15354.603} C_VEL
LIN {X 0,Y 307.21,Z 959.888,A -85,B 0,C 180,E1 15360.074,E2 15360.074} C_VEL
LIN {X 0,Y 300.433,Z 980.768,A -85,B 0,C 180,E1 15366.223,E2 15366.223} C_VEL
LIN {X 0,Y 296.336,Z 996.337,A -85,B 0,C 180,E1 15372.915,E2 15372.915} C_VEL
LIN {X 0,Y 294.706,Z 1006.374,A -85,B 0,C 180,E1 15379.64,E2 15379.64} C_VEL
LIN {X 0,Y 294.486,Z 1010.272,A -85,B 0,C 180,E1 15384.097,E2 15384.097} C_VEL
LIN {X 0,Y 294.529,Z 1012.209,A -85,B 0,C 180,E1 15390,E2 15390} C_VEL
LIN {X 0,Y 294.503,Z 1010.283,A -85,B 0,C 180,E1 15395.901,E2 15395.901} C_VEL
LIN {X 0,Y 295.146,Z 1003.135,A -85,B 0,C 180,E1 15402.96,E2 15402.96} C_VEL
LIN {X 0,Y 297.759,Z 990.348,A -85,B 0,C 180,E1 15410.016,E2 15410.016} C_VEL
LIN {X 0,Y 303.261,Z 971.784,A -85,B 0,C 180,E1 15416.701,E2 15416.701} C_VEL
LIN {X 0,Y 310.95,Z 949.145,A -85,B 0,C 180,E1 15422.385,E2 15422.385} C_VEL
LIN {X 0,Y 320.067,Z 922.13,A -85,B 0,C 180,E1 15427.201,E2 15427.201} C_VEL
LIN {X 0,Y 329.481,Z 890.68,A -85,B 0,C 180,E1 15431.125,E2 15431.125} C_VEL
LIN {X 0,Y 338.275,Z 855.692,A -85,B 0,C 180,E1 15434.045,E2 15434.045} C_VEL
LIN {X 0,Y 343.185,Z 831.889,A -85,B 0,C 180,E1 15435.477,E2 15435.477} C_VEL
LIN {X 0,Y 345.882,Z 820.398,A -85,B 0,C 180,E1 15437.334,E2 15437.334} C_VEL
LIN {X 0,Y 345.164,Z 819.11,A -85,B 0,C 180,E1 15438.439,E2 15438.439} C_VEL
LIN {X 0,Y 341.244,Z 823.188,A -85,B 0,C 180,E1 15441.171,E2 15441.171} C_VEL
LIN {X 0,Y 341.061,Z 824.542,A -85,B 0,C 180,E1 15442.907,E2 15442.907} C_VEL
LIN {X 0,Y 328.032,Z 854.521,A -85,B 0,C 180,E1 15446.376,E2 15446.376} C_VEL
LIN {X 0,Y 317.455,Z 877.21,A -85,B 0,C 180,E1 15450.35,E2 15450.35} C_VEL
LIN {X 0,Y 307.562,Z 895.748,A -85,B 0,C 180,E1 15455.272,E2 15455.272} C_VEL
LIN {X 0,Y 299.643,Z 908.431,A -85,B 0,C 180,E1 15460.834,E2 15460.834} C_VEL
LIN {X 0,Y 295.331,Z 913.944,A -85,B 0,C 180,E1 15465.155,E2 15465.155} C_VEL
LIN {X 0,Y 291.605,Z 916.444,A -85,B 0,C 180,E1 15471.046,E2 15471.046} C_VEL
LIN {X 0,Y 289.813,Z 913.4,A -85,B 0,C 180,E1 15477.012,E2 15477.012} C_VEL
LIN {X 0,Y 289.729,Z 904.651,A -85,B 0,C 180,E1 15483.002,E2 15483.002} C_VEL
LIN {X 0,Y 290.896,Z 890.624,A -85,B 0,C 180,E1 15488.533,E2 15488.533} C_VEL
LIN {X 0,Y 293.166,Z 871.857,A -85,B 0,C 180,E1 15493.445,E2 15493.445} C_VEL
LIN {X 0,Y 296.154,Z 848.291,A -85,B 0,C 180,E1 15497.677,E2 15497.677} C_VEL
LIN {X 0,Y 299.466,Z 819.68,A -85,B 0,C 180,E1 15501.121,E2 15501.121} C_VEL
LIN {X 0,Y 301.017,Z 790.934,A -85,B 0,C 180,E1 15503.374,E2 15503.374} C_VEL
LIN {X 0,Y 288.373,Z 747.293,A -85,B 0,C 180,E1 15506.573,E2 15506.573} C_VEL
LIN {X 0,Y 291.621,Z 745.849,A -85,B 0,C 180,E1 15507.758,E2 15507.758} C_VEL
LIN {X 0,Y 295.351,Z 750.815,A -85,B 0,C 180,E1 15509.36,E2 15509.36} C_VEL
LIN {X 0,Y 307.243,Z 768.122,A -85,B 0,C 180,E1 15513.887,E2 15513.887} C_VEL
LIN {X 0,Y 320.944,Z 793.245,A -85,B 0,C 180,E1 15518.91,E2 15518.91} C_VEL
LIN {X 0,Y 330.728,Z 818.648,A -85,B 0,C 180,E1 15523.128,E2 15523.128} C_VEL
LIN {X 0,Y 334.319,Z 833.721,A -85,B 0,C 180,E1 15525.378,E2 15525.378} C_VEL
LIN {X 0,Y 325.947,Z 866.893,A -85,B 0,C 180,E1 15528.366,E2 15528.366} C_VEL
LIN {X 0,Y 316.223,Z 897.341,A -85,B 0,C 180,E1 15532.36,E2 15532.36} C_VEL
LIN {X 0,Y 306.292,Z 924.437,A -85,B 0,C 180,E1 15537.481,E2 15537.481} C_VEL
LIN {X 0,Y 297.677,Z 946.812,A -85,B 0,C 180,E1 15543.574,E2 15543.574} C_VEL
LIN {X 0,Y 291.56,Z 963.427,A -85,B 0,C 180,E1 15550.273,E2 15550.273} C_VEL
LIN {X 0,Y 288.199,Z 974.255,A -85,B 0,C 180,E1 15556.961,E2 15556.961} C_VEL
LIN {X 0,Y 286.7,Z 980.546,A -85,B 0,C 180,E1 15563.937,E2 15563.937} C_VEL
LIN {X 0,Y 286.585,Z 982.279,A -85,B 0,C 180,E1 15570,E2 15570} C_VEL
LIN {X 0,Y 286.906,Z 979.51,A -85,B 0,C 180,E1 15577.582,E2 15577.582} C_VEL
LIN {X 0,Y 289.077,Z 971.171,A -85,B 0,C 180,E1 15585.182,E2 15585.182} C_VEL
LIN {X 0,Y 293.264,Z 958.503,A -85,B 0,C 180,E1 15591.902,E2 15591.902} C_VEL
LIN {X 0,Y 300.391,Z 939.581,A -85,B 0,C 180,E1 15598.548,E2 15598.548} C_VEL
LIN {X 0,Y 309.488,Z 915.816,A -85,B 0,C 180,E1 15604.249,E2 15604.249} C_VEL
LIN {X 0,Y 319.316,Z 888,A -85,B 0,C 180,E1 15608.923,E2 15608.923} C_VEL
LIN {X 0,Y 328.671,Z 856.737,A -85,B 0,C 180,E1 15612.573,E2 15612.573} C_VEL
LIN {X 0,Y 334.182,Z 832.012,A -85,B 0,C 180,E1 15614.716,E2 15614.716} C_VEL
LIN {X 0,Y 325.652,Z 804.401,A -85,B 0,C 180,E1 15619.054,E2 15619.054} C_VEL
LIN {X 0,Y 313.28,Z 778.311,A -85,B 0,C 180,E1 15623.8,E2 15623.8} C_VEL
LIN {X 0,Y 298.185,Z 754.207,A -85,B 0,C 180,E1 15629.361,E2 15629.361} C_VEL
LIN {X 0,Y 291.677,Z 745.899,A -85,B 0,C 180,E1 15632.047,E2 15632.047} C_VEL
LIN {X 0,Y 288.227,Z 740.492,A -85,B 0,C 180,E1 15633.684,E2 15633.684} C_VEL
LIN {X 0,Y 284.631,Z 735.674,A -85,B 0,C 180,E1 15635.494,E2 15635.494} C_VEL
LIN {X 0,Y 284.332,Z 733.66,A -85,B 0,C 180,E1 15635.829,E2 15635.829} C_VEL
LIN {X 0,Y 284.794,Z 733.66,A -85,B 0,C 180,E1 15644.578,E2 15644.578} C_VEL
LIN {X 0,Y 285.236,Z 733.66,A -85,B 0,C 180,E1 15651.76,E2 15651.76} C_VEL
LIN {X 0,Y 286.12,Z 733.66,A -85,B 0,C 180,E1 15659.993,E2 15659.993} C_VEL
LIN {X 0,Y 285.541,Z 733.66,A -85,B 0,C 180,E1 15666.081,E2 15666.081} C_VEL
LIN {X 0,Y 285.085,Z 733.66,A -85,B 0,C 180,E1 15672.258,E2 15672.258} C_VEL
LIN {X 0,Y 284.647,Z 733.66,A -85,B 0,C 180,E1 15678.603,E2 15678.603} C_VEL
LIN {X 0,Y 284.327,Z 733.969,A -85,B 0,C 180,E1 15683.739,E2 15683.739} C_VEL
LIN {X 0,Y 286.509,Z 739.148,A -85,B 0,C 180,E1 15685.001,E2 15685.001} C_VEL
LIN {X 0,Y 289.514,Z 741.933,A -85,B 0,C 180,E1 15686.384,E2 15686.384} C_VEL
LIN {X 0,Y 303.556,Z 762.485,A -85,B 0,C 180,E1 15692.157,E2 15692.157} C_VEL
LIN {X 0,Y 319.461,Z 788.068,A -85,B 0,C 180,E1 15697.381,E2 15697.381} C_VEL
LIN {X 0,Y 330.271,Z 810.708,A -85,B 0,C 180,E1 15700.89,E2 15700.89} C_VEL
LIN {X 0,Y 336.072,Z 838.131,A -85,B 0,C 180,E1 15703.979,E2 15703.979} C_VEL
LIN {X 0,Y 328.005,Z 873.808,A -85,B 0,C 180,E1 15706.407,E2 15706.407} C_VEL
LIN {X 0,Y 318.54,Z 906.399,A -85,B 0,C 180,E1 15709.804,E2 15709.804} C_VEL
LIN {X 0,Y 309.101,Z 934.4,A -85,B 0,C 180,E1 15713.998,E2 15713.998} C_VEL
LIN {X 0,Y 299.702,Z 960.9,A -85,B 0,C 180,E1 15719.655,E2 15719.655} C_VEL
LIN {X 0,Y 292.346,Z 982.342,A -85,B 0,C 180,E1 15726.335,E2 15726.335} C_VEL
LIN {X 0,Y 288.288,Z 997.298,A -85,B 0,C 180,E1 15733.21,E2 15733.21} C_VEL
LIN {X 0,Y 286.842,Z 1005.962,A -85,B 0,C 180,E1 15739.353,E2 15739.353} C_VEL
LIN {X 0,Y 286.611,Z 1009.864,A -85,B 0,C 180,E1 15743.935,E2 15743.935} C_VEL
LIN {X 0,Y 286.653,Z 1011.803,A -85,B 0,C 180,E1 15750,E2 15750} C_VEL
LIN {X 0,Y 286.626,Z 1009.875,A -85,B 0,C 180,E1 15756.064,E2 15756.064} C_VEL
LIN {X 0,Y 287.302,Z 1002.721,A -85,B 0,C 180,E1 15763.32,E2 15763.32} C_VEL
LIN {X 0,Y 290.149,Z 989.998,A -85,B 0,C 180,E1 15770.535,E2 15770.535} C_VEL
LIN {X 0,Y 296.02,Z 971.37,A -85,B 0,C 180,E1 15777.408,E2 15777.408} C_VEL
LIN {X 0,Y 304.11,Z 948.734,A -85,B 0,C 180,E1 15783.206,E2 15783.206} C_VEL
LIN {X 0,Y 314.231,Z 920.062,A -85,B 0,C 180,E1 15788.343,E2 15788.343} C_VEL
LIN {X 0,Y 323.946,Z 888.75,A -85,B 0,C 180,E1 15792.211,E2 15792.211} C_VEL
LIN {X 0,Y 332.727,Z 854.735,A -85,B 0,C 180,E1 15795.039,E2 15795.039} C_VEL
LIN {X 0,Y 336.5,Z 840.445,A -85,B 0,C 180,E1 15796.048,E2 15796.048} C_VEL
LIN {X 0,Y 339.888,Z 832.107,A -85,B 0,C 180,E1 15796.928,E2 15796.928} C_VEL
LIN {X 0,Y 342.099,Z 824.355,A -85,B 0,C 180,E1 15798.414,E2 15798.414} C_VEL
LIN {X 0,Y 341.244,Z 823.188,A -85,B 0,C 180,E1 15801.171,E2 15801.171} C_VEL
LIN {X 0,Y 339.807,Z 825.871,A -85,B 0,C 180,E1 15802.033,E2 15802.033} C_VEL
LIN {X 0,Y 331.848,Z 841.402,A -85,B 0,C 180,E1 15803.198,E2 15803.198} C_VEL
LIN {X 0,Y 318.385,Z 868.195,A -85,B 0,C 180,E1 15807.061,E2 15807.061} C_VEL
LIN {X 0,Y 306.195,Z 890.251,A -85,B 0,C 180,E1 15811.99,E2 15811.99} C_VEL
LIN {X 0,Y 296.409,Z 905.517,A -85,B 0,C 180,E1 15817.482,E2 15817.482} C_VEL
LIN {X 0,Y 289.369,Z 914.495,A -85,B 0,C 180,E1 15823.283,E2 15823.283} C_VEL
LIN {X 0,Y 285.583,Z 917.617,A -85,B 0,C 180,E1 15827.764,E2 15827.764} C_VEL
LIN {X 0,Y 282.815,Z 916.95,A -85,B 0,C 180,E1 15833.861,E2 15833.861} C_VEL
LIN {X 0,Y 281.751,Z 910.826,A -85,B 0,C 180,E1 15840.007,E2 15840.007} C_VEL
LIN {X 0,Y 282.368,Z 898.574,A -85,B 0,C 180,E1 15846.163,E2 15846.163} C_VEL
LIN {X 0,Y 284.277,Z 881.587,A -85,B 0,C 180,E1 15851.527,E2 15851.527} C_VEL
LIN {X 0,Y 287.118,Z 859.58,A -85,B 0,C 180,E1 15856.275,E2 15856.275} C_VEL
LIN {X 0,Y 290.421,Z 833.423,A -85,B 0,C 180,E1 15860.12,E2 15860.12} C_VEL
LIN {X 0,Y 293.473,Z 803.08,A -85,B 0,C 180,E1 15863.016,E2 15863.016} C_VEL
LIN {X 0,Y 293.122,Z 791.004,A -85,B 0,C 180,E1 15863.9,E2 15863.9} C_VEL
LIN {X 0,Y 285.128,Z 762.175,A -85,B 0,C 180,E1 15866.081,E2 15866.081} C_VEL
LIN {X 0,Y 287.559,Z 760.647,A -85,B 0,C 180,E1 15866.98,E2 15866.98} C_VEL
LIN {X 0,Y 290.72,Z 754.37,A -85,B 0,C 180,E1 15867.864,E2 15867.864} C_VEL
LIN {X 0,Y 304.473,Z 775.49,A -85,B 0,C 180,E1 15873.487,E2 15873.487} C_VEL
LIN {X 0,Y 317.185,Z 800.43,A -85,B 0,C 180,E1 15878.621,E2 15878.621} C_VEL
LIN {X 0,Y 326.203,Z 826.354,A -85,B 0,C 180,E1 15883.051,E2 15883.051} C_VEL
LIN {X 0,Y 328.085,Z 837.025,A -85,B 0,C 180,E1 15884.625,E2 15884.625} C_VEL
LIN {X 0,Y 318.771,Z 871.407,A -85,B 0,C 180,E1 15887.888,E2 15887.888} C_VEL
LIN {X 0,Y 308.601,Z 901.295,A -85,B 0,C 180,E1 15892.036,E2 15892.036} C_VEL
LIN {X 0,Y 298.318,Z 928.122,A -85,B 0,C 180,E1 15897.427,E2 15897.427} C_VEL
LIN {X 0,Y 289.649,Z 949.329,A -85,B 0,C 180,E1 15903.62,E2 15903.62} C_VEL
LIN {X 0,Y 283.488,Z 965.36,A -85,B 0,C 180,E1 15910.524,E2 15910.524} C_VEL
LIN {X 0,Y 280.162,Z 975.754,A -85,B 0,C 180,E1 15917.516,E2 15917.516} C_VEL
LIN {X 0,Y 278.826,Z 980.954,A -85,B 0,C 180,E1 15923.766,E2 15923.766} C_VEL
LIN {X 0,Y 278.693,Z 982.685,A -85,B 0,C 180,E1 15930,E2 15930} C_VEL
LIN {X 0,Y 279.064,Z 979.918,A -85,B 0,C 180,E1 15937.796,E2 15937.796} C_VEL
LIN {X 0,Y 281.378,Z 971.583,A -85,B 0,C 180,E1 15945.608,E2 15945.608} C_VEL
LIN {X 0,Y 285.946,Z 958.744,A -85,B 0,C 180,E1 15952.575,E2 15952.575} C_VEL
LIN {X 0,Y 293.455,Z 939.803,A -85,B 0,C 180,E1 15959.35,E2 15959.35} C_VEL
LIN {X 0,Y 302.93,Z 916.272,A -85,B 0,C 180,E1 15965.085,E2 15965.085} C_VEL
LIN {X 0,Y 313.191,Z 888.401,A -85,B 0,C 180,E1 15969.834,E2 15969.834} C_VEL
LIN {X 0,Y 323.139,Z 856.165,A -85,B 0,C 180,E1 15973.615,E2 15973.615} C_VEL
LIN {X 0,Y 328.137,Z 835.1,A -85,B 0,C 180,E1 15975.464,E2 15975.464} C_VEL
LIN {X 0,Y 320.582,Z 809.191,A -85,B 0,C 180,E1 15979.715,E2 15979.715} C_VEL
LIN {X 0,Y 308.916,Z 783.29,A -85,B 0,C 180,E1 15984.617,E2 15984.617} C_VEL
LIN {X 0,Y 294.798,Z 760.37,A -85,B 0,C 180,E1 15990.204,E2 15990.204} C_VEL
LIN {X 0,Y 285.186,Z 747.117,A -85,B 0,C 180,E1 15994.575,E2 15994.575} C_VEL
LIN {X 0,Y 281.005,Z 740.791,A -85,B 0,C 180,E1 15996.861,E2 15996.861} C_VEL
LIN {X 0,Y 276.916,Z 736.18,A -85,B 0,C 180,E1 15999.29,E2 15999.29} C_VEL
LIN {X 0,Y 276.515,Z 733.66,A -85,B 0,C 180,E1 15999.779,E2 15999.779} C_VEL
LIN {X 0,Y 277.035,Z 733.66,A -85,B 0,C 180,E1 16007.366,E2 16007.366} C_VEL
LIN {X 0,Y 277.94,Z 733.66,A -85,B 0,C 180,E1 16016.87,E2 16016.87} C_VEL
LIN {X 0,Y 277.946,Z 733.66,A -85,B 0,C 180,E1 16023.116,E2 16023.116} C_VEL
LIN {X 0,Y 277.113,Z 733.66,A -85,B 0,C 180,E1 16032.616,E2 16032.616} C_VEL
LIN {X 0,Y 276.581,Z 733.835,A -85,B 0,C 180,E1 16039.823,E2 16039.823} C_VEL
LIN {X 0,Y 278.35,Z 738.68,A -85,B 0,C 180,E1 16041.135,E2 16041.135} C_VEL
LIN {X 0,Y 282.089,Z 742.377,A -85,B 0,C 180,E1 16043.228,E2 16043.228} C_VEL
LIN {X 0,Y 288.437,Z 751.743,A -85,B 0,C 180,E1 16046.49,E2 16046.49} C_VEL
LIN {X 0,Y 297.546,Z 764.62,A -85,B 0,C 180,E1 16050.386,E2 16050.386} C_VEL
LIN {X 0,Y 312.139,Z 787.639,A -85,B 0,C 180,E1 16055.587,E2 16055.587} C_VEL
LIN {X 0,Y 324.777,Z 813.473,A -85,B 0,C 180,E1 16059.966,E2 16059.966} C_VEL
LIN {X 0,Y 330.195,Z 839.829,A -85,B 0,C 180,E1 16063.092,E2 16063.092} C_VEL
LIN {X 0,Y 321.775,Z 875.118,A -85,B 0,C 180,E1 16065.578,E2 16065.578} C_VEL
LIN {X 0,Y 312.304,Z 906.424,A -85,B 0,C 180,E1 16068.909,E2 16068.909} C_VEL
LIN {X 0,Y 301.801,Z 936.218,A -85,B 0,C 180,E1 16073.5,E2 16073.5} C_VEL
LIN {X 0,Y 292.18,Z 961.835,A -85,B 0,C 180,E1 16079.22,E2 16079.22} C_VEL
LIN {X 0,Y 284.933,Z 981.925,A -85,B 0,C 180,E1 16085.68,E2 16085.68} C_VEL
LIN {X 0,Y 280.555,Z 996.881,A -85,B 0,C 180,E1 16092.733,E2 16092.733} C_VEL
LIN {X 0,Y 278.998,Z 1005.55,A -85,B 0,C 180,E1 16099.05,E2 16099.05} C_VEL
LIN {X 0,Y 278.713,Z 1009.455,A -85,B 0,C 180,E1 16103.762,E2 16103.762} C_VEL
LIN {X 0,Y 278.759,Z 1011.396,A -85,B 0,C 180,E1 16110,E2 16110} C_VEL
LIN {X 0,Y 278.728,Z 1009.467,A -85,B 0,C 180,E1 16116.237,E2 16116.237} C_VEL
LIN {X 0,Y 279.265,Z 1003.637,A -85,B 0,C 180,E1 16122.649,E2 16122.649} C_VEL
LIN {X 0,Y 281.739,Z 992.534,A -85,B 0,C 180,E1 16129.648,E2 16129.648} C_VEL
LIN {X 0,Y 286.993,Z 976.15,A -85,B 0,C 180,E1 16136.443,E2 16136.443} C_VEL
LIN {X 0,Y 295.267,Z 953.848,A -85,B 0,C 180,E1 16142.816,E2 16142.816} C_VEL
LIN {X 0,Y 305.652,Z 926.091,A -85,B 0,C 180,E1 16148.258,E2 16148.258} C_VEL
LIN {X 0,Y 315.782,Z 895.721,A -85,B 0,C 180,E1 16152.396,E2 16152.396} C_VEL
LIN {X 0,Y 325.716,Z 860.399,A -85,B 0,C 180,E1 16155.612,E2 16155.612} C_VEL
LIN {X 0,Y 330.203,Z 848.28,A -85,B 0,C 180,E1 16156.665,E2 16156.665} C_VEL
LIN {X 0,Y 336.026,Z 835.965,A -85,B 0,C 180,E1 16157.893,E2 16157.893} C_VEL
LIN {X 0,Y 337.95,Z 830.873,A -85,B 0,C 180,E1 16158.808,E2 16158.808} C_VEL
LIN {X 0,Y 337.334,Z 830.237,A -85,B 0,C 180,E1 16161.901,E2 16161.901} C_VEL
LIN {X 0,Y 331.848,Z 841.402,A -85,B 0,C 180,E1 16163.198,E2 16163.198} C_VEL
LIN {X 0,Y 317.032,Z 865.961,A -85,B 0,C 180,E1 16165.143,E2 16165.143} C_VEL
LIN {X 0,Y 315.207,Z 868.925,A -85,B 0,C 180,E1 16165.603,E2 16165.603} C_VEL
LIN {X 0,Y 302.173,Z 890.314,A -85,B 0,C 180,E1 16170.352,E2 16170.352} C_VEL
LIN {X 0,Y 291.849,Z 905.167,A -85,B 0,C 180,E1 16175.487,E2 16175.487} C_VEL
LIN {X 0,Y 283.675,Z 914.989,A -85,B 0,C 180,E1 16181.331,E2 16181.331} C_VEL
LIN {X 0,Y 278.054,Z 919.353,A -85,B 0,C 180,E1 16187.427,E2 16187.427} C_VEL
LIN {X 0,Y 275.065,Z 918.295,A -85,B 0,C 180,E1 16193.687,E2 16193.687} C_VEL
LIN {X 0,Y 273.931,Z 911.803,A -85,B 0,C 180,E1 16200.007,E2 16200.007} C_VEL
LIN {X 0,Y 274.554,Z 899.208,A -85,B 0,C 180,E1 16206.339,E2 16206.339} C_VEL
LIN {X 0,Y 276.543,Z 881.922,A -85,B 0,C 180,E1 16211.854,E2 16211.854} C_VEL
LIN {X 0,Y 279.503,Z 859.411,A -85,B 0,C 180,E1 16216.732,E2 16216.732} C_VEL
LIN {X 0,Y 282.961,Z 832.727,A -85,B 0,C 180,E1 16220.674,E2 16220.674} C_VEL
LIN {X 0,Y 286.036,Z 802.823,A -85,B 0,C 180,E1 16223.555,E2 16223.555} C_VEL
LIN {X 0,Y 285.524,Z 792.077,A -85,B 0,C 180,E1 16224.368,E2 16224.368} C_VEL
LIN {X 0,Y 281.75,Z 777.025,A -85,B 0,C 180,E1 16225.664,E2 16225.664} C_VEL
LIN {X 0,Y 284.573,Z 774.464,A -85,B 0,C 180,E1 16226.66,E2 16226.66} C_VEL
LIN {X 0,Y 287.533,Z 768.688,A -85,B 0,C 180,E1 16227.442,E2 16227.442} C_VEL
LIN {X 0,Y 290.62,Z 765.187,A -85,B 0,C 180,E1 16228.391,E2 16228.391} C_VEL
LIN {X 0,Y 302.474,Z 784.412,A -85,B 0,C 180,E1 16233.523,E2 16233.523} C_VEL
LIN {X 0,Y 313.728,Z 808.877,A -85,B 0,C 180,E1 16238.567,E2 16238.567} C_VEL
LIN {X 0,Y 321.154,Z 833.075,A -85,B 0,C 180,E1 16242.825,E2 16242.825} C_VEL
LIN {X 0,Y 321.738,Z 840.865,A -85,B 0,C 180,E1 16243.902,E2 16243.902} C_VEL
LIN {X 0,Y 312.103,Z 874.372,A -85,B 0,C 180,E1 16247.221,E2 16247.221} C_VEL
LIN {X 0,Y 301.161,Z 904.949,A -85,B 0,C 180,E1 16251.659,E2 16251.659} C_VEL
LIN {X 0,Y 290.722,Z 930.495,A -85,B 0,C 180,E1 16257.083,E2 16257.083} C_VEL
LIN {X 0,Y 282.407,Z 949.972,A -85,B 0,C 180,E1 16262.986,E2 16262.986} C_VEL
LIN {X 0,Y 275.883,Z 966.008,A -85,B 0,C 180,E1 16270.099,E2 16270.099} C_VEL
LIN {X 0,Y 272.396,Z 976.162,A -85,B 0,C 180,E1 16277.154,E2 16277.154} C_VEL
LIN {X 0,Y 270.978,Z 981.36,A -85,B 0,C 180,E1 16283.584,E2 16283.584} C_VEL
LIN {X 0,Y 270.816,Z 983.091,A -85,B 0,C 180,E1 16290,E2 16290} C_VEL
LIN {X 0,Y 271.23,Z 980.326,A -85,B 0,C 180,E1 16298.023,E2 16298.023} C_VEL
LIN {X 0,Y 273.7,Z 971.994,A -85,B 0,C 180,E1 16306.058,E2 16306.058} C_VEL
LIN {X 0,Y 278.574,Z 959.156,A -85,B 0,C 180,E1 16313.207,E2 16313.207} C_VEL
LIN {X 0,Y 286.498,Z 940.209,A -85,B 0,C 180,E1 16320.137,E2 16320.137} C_VEL
LIN {X 0,Y 296.425,Z 916.681,A -85,B 0,C 180,E1 16325.973,E2 16325.973} C_VEL
LIN {X 0,Y 307.138,Z 888.803,A -85,B 0,C 180,E1 16330.783,E2 16330.783} C_VEL
LIN {X 0,Y 317.351,Z 856.888,A -85,B 0,C 180,E1 16334.572,E2 16334.572} C_VEL
LIN {X 0,Y 322.091,Z 837.834,A -85,B 0,C 180,E1 16336.293,E2 16336.293} C_VEL
LIN {X 0,Y 314.573,Z 811.663,A -85,B 0,C 180,E1 16340.817,E2 16340.817} C_VEL
LIN {X 0,Y 304.326,Z 788.123,A -85,B 0,C 180,E1 16345.527,E2 16345.527} C_VEL
LIN {X 0,Y 291.86,Z 766.86,A -85,B 0,C 180,E1 16350.893,E2 16350.893} C_VEL
LIN {X 0,Y 282.543,Z 753.833,A -85,B 0,C 180,E1 16355.333,E2 16355.333} C_VEL
LIN {X 0,Y 278.34,Z 747.776,A -85,B 0,C 180,E1 16357.721,E2 16357.721} C_VEL
LIN {X 0,Y 274.439,Z 742.006,A -85,B 0,C 180,E1 16360.272,E2 16360.272} C_VEL
LIN {X 0,Y 269.423,Z 736.402,A -85,B 0,C 180,E1 16364.093,E2 16364.093} C_VEL
LIN {X 0,Y 268.918,Z 733.66,A -85,B 0,C 180,E1 16364.899,E2 16364.899} C_VEL
LIN {X 0,Y 269.637,Z 733.66,A -85,B 0,C 180,E1 16373.545,E2 16373.545} C_VEL
LIN {X 0,Y 270.326,Z 733.66,A -85,B 0,C 180,E1 16379.993,E2 16379.993} C_VEL
LIN {X 0,Y 269.671,Z 733.66,A -85,B 0,C 180,E1 16386.44,E2 16386.44} C_VEL
LIN {X 0,Y 269.018,Z 734.413,A -85,B 0,C 180,E1 16394.871,E2 16394.871} C_VEL
LIN {X 0,Y 271.797,Z 739.876,A -85,B 0,C 180,E1 16397.377,E2 16397.377} C_VEL
LIN {X 0,Y 274.479,Z 741.987,A -85,B 0,C 180,E1 16399.222,E2 16399.222} C_VEL
LIN {X 0,Y 278.229,Z 747.636,A -85,B 0,C 180,E1 16401.685,E2 16401.685} C_VEL
LIN {X 0,Y 280.879,Z 751.548,A -85,B 0,C 180,E1 16403.236,E2 16403.236} C_VEL
LIN {X 0,Y 286.502,Z 759.325,A -85,B 0,C 180,E1 16406.134,E2 16406.134} C_VEL
LIN {X 0,Y 297.985,Z 776.223,A -85,B 0,C 180,E1 16411.058,E2 16411.058} C_VEL
LIN {X 0,Y 311.978,Z 800.595,A -85,B 0,C 180,E1 16416.252,E2 16416.252} C_VEL
LIN {X 0,Y 320.404,Z 820.761,A -85,B 0,C 180,E1 16419.588,E2 16419.588} C_VEL
LIN {X 0,Y 323.947,Z 843.191,A -85,B 0,C 180,E1 16422.277,E2 16422.277} C_VEL
LIN {X 0,Y 315.113,Z 878.132,A -85,B 0,C 180,E1 16424.868,E2 16424.868} C_VEL
LIN {X 0,Y 304.562,Z 910.994,A -85,B 0,C 180,E1 16428.565,E2 16428.565} C_VEL
LIN {X 0,Y 294.144,Z 938.961,A -85,B 0,C 180,E1 16433.181,E2 16433.181} C_VEL
LIN {X 0,Y 284.69,Z 962.767,A -85,B 0,C 180,E1 16438.765,E2 16438.765} C_VEL
LIN {X 0,Y 276.845,Z 983.499,A -85,B 0,C 180,E1 16445.783,E2 16445.783} C_VEL
LIN {X 0,Y 272.521,Z 997.827,A -85,B 0,C 180,E1 16453.041,E2 16453.041} C_VEL
LIN {X 0,Y 270.945,Z 1006.729,A -85,B 0,C 180,E1 16460.349,E2 16460.349} C_VEL
LIN {X 0,Y 270.749,Z 1010.463,A -85,B 0,C 180,E1 16466.794,E2 16466.794} C_VEL
LIN {X 0,Y 270.788,Z 1010.471,A -85,B 0,C 180,E1 16473.205,E2 16473.205} C_VEL
LIN {X 0,Y 270.967,Z 1006.746,A -85,B 0,C 180,E1 16479.65,E2 16479.65} C_VEL
LIN {X 0,Y 272.581,Z 997.855,A -85,B 0,C 180,E1 16486.954,E2 16486.954} C_VEL
LIN {X 0,Y 276.923,Z 983.555,A -85,B 0,C 180,E1 16494.209,E2 16494.209} C_VEL
LIN {X 0,Y 284.708,Z 962.843,A -85,B 0,C 180,E1 16501.232,E2 16501.232} C_VEL
LIN {X 0,Y 294.895,Z 937.241,A -85,B 0,C 180,E1 16507.181,E2 16507.181} C_VEL
LIN {X 0,Y 305.844,Z 907.676,A -85,B 0,C 180,E1 16511.874,E2 16511.874} C_VEL
LIN {X 0,Y 315.718,Z 876.666,A -85,B 0,C 180,E1 16515.264,E2 16515.264} C_VEL
LIN {X 0,Y 320.624,Z 862.13,A -85,B 0,C 180,E1 16516.637,E2 16516.637} C_VEL
LIN {X 0,Y 332.642,Z 839.584,A -85,B 0,C 180,E1 16518.951,E2 16518.951} C_VEL
LIN {X 0,Y 333.203,Z 838.367,A -85,B 0,C 180,E1 16519.163,E2 16519.163} C_VEL
LIN {X 0,Y 333.391,Z 836.952,A -85,B 0,C 180,E1 16520.538,E2 16520.538} C_VEL
LIN {X 0,Y 332.971,Z 837.601,A -85,B 0,C 180,E1 16521.257,E2 16521.257} C_VEL
LIN {X 0,Y 317.062,Z 865.731,A -85,B 0,C 180,E1 16525.047,E2 16525.047} C_VEL
LIN {X 0,Y 315.207,Z 868.925,A -85,B 0,C 180,E1 16525.603,E2 16525.603} C_VEL
LIN {X 0,Y 306.345,Z 881.308,A -85,B 0,C 180,E1 16527.257,E2 16527.257} C_VEL
LIN {X 0,Y 298.279,Z 891.12,A -85,B 0,C 180,E1 16528.84,E2 16528.84} C_VEL
LIN {X 0,Y 297.393,Z 892.288,A -85,B 0,C 180,E1 16529.147,E2 16529.147} C_VEL
LIN {X 0,Y 285.187,Z 908.05,A -85,B 0,C 180,E1 16534.875,E2 16534.875} C_VEL
LIN {X 0,Y 276.514,Z 917.221,A -85,B 0,C 180,E1 16540.828,E2 16540.828} C_VEL
LIN {X 0,Y 270.519,Z 921.058,A -85,B 0,C 180,E1 16547.071,E2 16547.071} C_VEL
LIN {X 0,Y 267.314,Z 919.636,A -85,B 0,C 180,E1 16553.503,E2 16553.503} C_VEL
LIN {X 0,Y 266.093,Z 912.734,A -85,B 0,C 180,E1 16560.007,E2 16560.007} C_VEL
LIN {X 0,Y 266.664,Z 900.825,A -85,B 0,C 180,E1 16566.118,E2 16566.118} C_VEL
LIN {X 0,Y 268.802,Z 882.128,A -85,B 0,C 180,E1 16572.201,E2 16572.201} C_VEL
LIN {X 0,Y 271.907,Z 859.24,A -85,B 0,C 180,E1 16577.213,E2 16577.213} C_VEL
LIN {X 0,Y 275.457,Z 832.349,A -85,B 0,C 180,E1 16581.201,E2 16581.201} C_VEL
LIN {X 0,Y 278.575,Z 802.505,A -85,B 0,C 180,E1 16584.092,E2 16584.092} C_VEL
LIN {X 0,Y 277.831,Z 792.785,A -85,B 0,C 180,E1 16584.865,E2 16584.865} C_VEL
LIN {X 0,Y 277.464,Z 790.923,A -85,B 0,C 180,E1 16585.136,E2 16585.136} C_VEL
LIN {X 0,Y 280.283,Z 788.961,A -85,B 0,C 180,E1 16586.148,E2 16586.148} C_VEL
LIN {X 0,Y 283.845,Z 783.052,A -85,B 0,C 180,E1 16587.076,E2 16587.076} C_VEL
LIN {X 0,Y 289.395,Z 774.388,A -85,B 0,C 180,E1 16588.522,E2 16588.522} C_VEL
LIN {X 0,Y 300.343,Z 793.998,A -85,B 0,C 180,E1 16593.684,E2 16593.684} C_VEL
LIN {X 0,Y 309.953,Z 817.167,A -85,B 0,C 180,E1 16598.53,E2 16598.53} C_VEL
LIN {X 0,Y 316.119,Z 840.803,A -85,B 0,C 180,E1 16602.77,E2 16602.77} C_VEL
LIN {X 0,Y 306.89,Z 873.08,A -85,B 0,C 180,E1 16606.011,E2 16606.011} C_VEL
LIN {X 0,Y 295.869,Z 902.956,A -85,B 0,C 180,E1 16610.287,E2 16610.287} C_VEL
LIN {X 0,Y 284.775,Z 929.325,A -85,B 0,C 180,E1 16615.796,E2 16615.796} C_VEL
LIN {X 0,Y 275.053,Z 950.916,A -85,B 0,C 180,E1 16622.428,E2 16622.428} C_VEL
LIN {X 0,Y 267.913,Z 967.603,A -85,B 0,C 180,E1 16630.179,E2 16630.179} C_VEL
LIN {X 0,Y 264.118,Z 978.201,A -85,B 0,C 180,E1 16638.426,E2 16638.426} C_VEL
LIN {X 0,Y 262.842,Z 983.049,A -85,B 0,C 180,E1 16646.698,E2 16646.698} C_VEL
LIN {X 0,Y 262.899,Z 983.011,A -85,B 0,C 180,E1 16653.302,E2 16653.302} C_VEL
LIN {X 0,Y 264.111,Z 978.1,A -85,B 0,C 180,E1 16661.575,E2 16661.575} C_VEL
LIN {X 0,Y 267.964,Z 967.419,A -85,B 0,C 180,E1 16669.818,E2 16669.818} C_VEL
LIN {X 0,Y 274.425,Z 952.279,A -85,B 0,C 180,E1 16676.947,E2 16676.947} C_VEL
LIN {X 0,Y 283.472,Z 932.055,A -85,B 0,C 180,E1 16683.379,E2 16683.379} C_VEL
LIN {X 0,Y 294.507,Z 906.317,A -85,B 0,C 180,E1 16689.005,E2 16689.005} C_VEL
LIN {X 0,Y 305.577,Z 876.788,A -85,B 0,C 180,E1 16693.432,E2 16693.432} C_VEL
LIN {X 0,Y 315.231,Z 845.054,A -85,B 0,C 180,E1 16696.696,E2 16696.696} C_VEL
LIN {X 0,Y 315.846,Z 839.61,A -85,B 0,C 180,E1 16697.323,E2 16697.323} C_VEL
LIN {X 0,Y 308.764,Z 814.12,A -85,B 0,C 180,E1 16701.944,E2 16701.944} C_VEL
LIN {X 0,Y 298.476,Z 790.204,A -85,B 0,C 180,E1 16707.056,E2 16707.056} C_VEL
LIN {X 0,Y 285.921,Z 768.502,A -85,B 0,C 180,E1 16713.03,E2 16713.03} C_VEL
LIN {X 0,Y 276.002,Z 754.801,A -85,B 0,C 180,E1 16718.456,E2 16718.456} C_VEL
LIN {X 0,Y 271.491,Z 748.317,A -85,B 0,C 180,E1 16721.584,E2 16721.584} C_VEL
LIN {X 0,Y 267.609,Z 743.298,A -85,B 0,C 180,E1 16724.824,E2 16724.824} C_VEL
LIN {X 0,Y 266.46,Z 741.157,A -85,B 0,C 180,E1 16726.018,E2 16726.018} C_VEL
LIN {X 0,Y 261.871,Z 736.077,A -85,B 0,C 180,E1 16731.996,E2 16731.996} C_VEL
LIN {X 0,Y 261.688,Z 733.66,A -85,B 0,C 180,E1 16733.348,E2 16733.348} C_VEL
LIN {X 0,Y 262.418,Z 733.66,A -85,B 0,C 180,E1 16739.993,E2 16739.993} C_VEL
LIN {X 0,Y 261.719,Z 734.256,A -85,B 0,C 180,E1 16746.845,E2 16746.845} C_VEL
LIN {X 0,Y 263.602,Z 739.142,A -85,B 0,C 180,E1 16750.332,E2 16750.332} C_VEL
LIN {X 0,Y 267.354,Z 742.293,A -85,B 0,C 180,E1 16754.337,E2 16754.337} C_VEL
LIN {X 0,Y 270.858,Z 747.896,A -85,B 0,C 180,E1 16757.439,E2 16757.439} C_VEL
LIN {X 0,Y 272.925,Z 750.383,A -85,B 0,C 180,E1 16758.947,E2 16758.947} C_VEL
LIN {X 0,Y 278.691,Z 758.577,A -85,B 0,C 180,E1 16762.639,E2 16762.639} C_VEL
LIN {X 0,Y 287.406,Z 771.006,A -85,B 0,C 180,E1 16767.122,E2 16767.122} C_VEL
LIN {X 0,Y 300.173,Z 791.401,A -85,B 0,C 180,E1 16772.504,E2 16772.504} C_VEL
LIN {X 0,Y 312.763,Z 817.304,A -85,B 0,C 180,E1 16777.615,E2 16777.615} C_VEL
LIN {X 0,Y 316.33,Z 831.133,A -85,B 0,C 180,E1 16779.608,E2 16779.608} C_VEL
LIN {X 0,Y 318.151,Z 845,A -85,B 0,C 180,E1 16781.35,E2 16781.35} C_VEL
LIN {X 0,Y 308.507,Z 881.147,A -85,B 0,C 180,E1 16784.129,E2 16784.129} C_VEL
LIN {X 0,Y 297.301,Z 913.943,A -85,B 0,C 180,E1 16788.029,E2 16788.029} C_VEL
LIN {X 0,Y 286.523,Z 941.444,A -85,B 0,C 180,E1 16792.811,E2 16792.811} C_VEL
LIN {X 0,Y 276.032,Z 966.55,A -85,B 0,C 180,E1 16799.115,E2 16799.115} C_VEL
LIN {X 0,Y 268.757,Z 984.951,A -85,B 0,C 180,E1 16805.892,E2 16805.892} C_VEL
LIN {X 0,Y 264.476,Z 998.6,A -85,B 0,C 180,E1 16813.366,E2 16813.366} C_VEL
LIN {X 0,Y 263.068,Z 1006.317,A -85,B 0,C 180,E1 16820.057,E2 16820.057} C_VEL
LIN {X 0,Y 262.846,Z 1010.055,A -85,B 0,C 180,E1 16826.697,E2 16826.697} C_VEL
LIN {X 0,Y 262.883,Z 1010.064,A -85,B 0,C 180,E1 16833.301,E2 16833.301} C_VEL
LIN {X 0,Y 263.091,Z 1006.335,A -85,B 0,C 180,E1 16839.941,E2 16839.941} C_VEL
LIN {X 0,Y 264.861,Z 997.441,A -85,B 0,C 180,E1 16847.464,E2 16847.464} C_VEL
LIN {X 0,Y 269.529,Z 983.14,A -85,B 0,C 180,E1 16854.917,E2 16854.917} C_VEL
LIN {X 0,Y 277.686,Z 962.715,A -85,B 0,C 180,E1 16862.018,E2 16862.018} C_VEL
LIN {X 0,Y 288.206,Z 937.52,A -85,B 0,C 180,E1 16868.014,E2 16868.014} C_VEL
LIN {X 0,Y 299.81,Z 907.535,A -85,B 0,C 180,E1 16872.867,E2 16872.867} C_VEL
LIN {X 0,Y 311.874,Z 873.253,A -85,B 0,C 180,E1 16876.737,E2 16876.737} C_VEL
LIN {X 0,Y 329.103,Z 844.415,A -85,B 0,C 180,E1 16879.913,E2 16879.913} C_VEL
LIN {X 0,Y 329.214,Z 844.006,A -85,B 0,C 180,E1 16880.331,E2 16880.331} C_VEL
LIN {X 0,Y 309.65,Z 874.377,A -85,B 0,C 180,E1 16884.943,E2 16884.943} C_VEL
LIN {X 0,Y 297.393,Z 892.288,A -85,B 0,C 180,E1 16889.147,E2 16889.147} C_VEL
LIN {X 0,Y 288.166,Z 902.132,A -85,B 0,C 180,E1 16891.379,E2 16891.379} C_VEL
LIN {X 0,Y 280.024,Z 909.446,A -85,B 0,C 180,E1 16893.509,E2 16893.509} C_VEL
LIN {X 0,Y 279.216,Z 910.256,A -85,B 0,C 180,E1 16893.885,E2 16893.885} C_VEL
LIN {X 0,Y 269.368,Z 919.463,A -85,B 0,C 180,E1 16900.299,E2 16900.299} C_VEL
LIN {X 0,Y 263.022,Z 922.768,A -85,B 0,C 180,E1 16906.696,E2 16906.696} C_VEL
LIN {X 0,Y 259.572,Z 920.929,A -85,B 0,C 180,E1 16913.308,E2 16913.308} C_VEL
LIN {X 0,Y 258.274,Z 913.667,A -85,B 0,C 180,E1 16920.008,E2 16920.008} C_VEL
LIN {X 0,Y 258.783,Z 902.237,A -85,B 0,C 180,E1 16925.939,E2 16925.939} C_VEL
LIN {X 0,Y 260.879,Z 883.798,A -85,B 0,C 180,E1 16932.152,E2 16932.152} C_VEL
LIN {X 0,Y 264.054,Z 861.046,A -85,B 0,C 180,E1 16937.311,E2 16937.311} C_VEL
LIN {X 0,Y 267.719,Z 834.278,A -85,B 0,C 180,E1 16941.464,E2 16941.464} C_VEL
LIN {X 0,Y 270.922,Z 807.572,A -85,B 0,C 180,E1 16944.347,E2 16944.347} C_VEL
LIN {X 0,Y 274.704,Z 803.586,A -85,B 0,C 180,E1 16945.512,E2 16945.512} C_VEL
LIN {X 0,Y 278.59,Z 797.593,A -85,B 0,C 180,E1 16946.428,E2 16946.428} C_VEL
LIN {X 0,Y 283.635,Z 790.973,A -85,B 0,C 180,E1 16947.744,E2 16947.744} C_VEL
LIN {X 0,Y 288.605,Z 784.646,A -85,B 0,C 180,E1 16949.037,E2 16949.037} C_VEL
LIN {X 0,Y 299.332,Z 806.748,A -85,B 0,C 180,E1 16954.628,E2 16954.628} C_VEL
LIN {X 0,Y 307.762,Z 831.806,A -85,B 0,C 180,E1 16959.764,E2 16959.764} C_VEL
LIN {X 0,Y 310.198,Z 844.344,A -85,B 0,C 180,E1 16962.024,E2 16962.024} C_VEL
LIN {X 0,Y 299.712,Z 877.872,A -85,B 0,C 180,E1 16965.498,E2 16965.498} C_VEL
LIN {X 0,Y 288.181,Z 907.197,A -85,B 0,C 180,E1 16969.967,E2 16969.967} C_VEL
LIN {X 0,Y 276.873,Z 932.471,A -85,B 0,C 180,E1 16975.598,E2 16975.598} C_VEL
LIN {X 0,Y 267.076,Z 953.265,A -85,B 0,C 180,E1 16982.378,E2 16982.378} C_VEL
LIN {X 0,Y 259.852,Z 969.305,A -85,B 0,C 180,E1 16990.426,E2 16990.426} C_VEL
LIN {X 0,Y 256.307,Z 978.666,A -85,B 0,C 180,E1 16998.133,E2 16998.133} C_VEL
LIN {X 0,Y 254.951,Z 983.456,A -85,B 0,C 180,E1 17006.596,E2 17006.596} C_VEL
LIN {X 0,Y 255.024,Z 983.418,A -85,B 0,C 180,E1 17013.404,E2 17013.404} C_VEL
LIN {X 0,Y 256.299,Z 978.573,A -85,B 0,C 180,E1 17021.861,E2 17021.861} C_VEL
LIN {X 0,Y 259.893,Z 969.137,A -85,B 0,C 180,E1 17029.572,E2 17029.572} C_VEL
LIN {X 0,Y 267.215,Z 952.907,A -85,B 0,C 180,E1 17037.642,E2 17037.642} C_VEL
LIN {X 0,Y 277.118,Z 931.865,A -85,B 0,C 180,E1 17044.448,E2 17044.448} C_VEL
LIN {X 0,Y 288.521,Z 906.394,A -85,B 0,C 180,E1 17050.06,E2 17050.06} C_VEL
LIN {X 0,Y 300.305,Z 875.829,A -85,B 0,C 180,E1 17054.645,E2 17054.645} C_VEL
LIN {X 0,Y 310.179,Z 844.297,A -85,B 0,C 180,E1 17057.856,E2 17057.856} C_VEL
LIN {X 0,Y 303.879,Z 819.129,A -85,B 0,C 180,E1 17062.625,E2 17062.625} C_VEL
LIN {X 0,Y 294.208,Z 795.512,A -85,B 0,C 180,E1 17067.902,E2 17067.902} C_VEL
LIN {X 0,Y 282.944,Z 774.957,A -85,B 0,C 180,E1 17073.796,E2 17073.796} C_VEL
LIN {X 0,Y 273.823,Z 761.792,A -85,B 0,C 180,E1 17079.141,E2 17079.141} C_VEL
LIN {X 0,Y 269.446,Z 755.588,A -85,B 0,C 180,E1 17082.315,E2 17082.315} C_VEL
LIN {X 0,Y 265.742,Z 749.836,A -85,B 0,C 180,E1 17085.687,E2 17085.687} C_VEL
LIN {X 0,Y 260.53,Z 742.943,A -85,B 0,C 180,E1 17092.834,E2 17092.834} C_VEL
LIN {X 0,Y 260.07,Z 741.389,A -85,B 0,C 180,E1 17094.145,E2 17094.145} C_VEL
LIN {X 0,Y 260.45,Z 741.459,A -85,B 0,C 180,E1 17106.145,E2 17106.145} C_VEL
LIN {X 0,Y 262.34,Z 746.755,A -85,B 0,C 180,E1 17109.963,E2 17109.963} C_VEL
LIN {X 0,Y 265.848,Z 750.015,A -85,B 0,C 180,E1 17113.894,E2 17113.894} C_VEL
LIN {X 0,Y 269.966,Z 755.863,A -85,B 0,C 180,E1 17117.528,E2 17117.528} C_VEL
LIN {X 0,Y 276.94,Z 766.232,A -85,B 0,C 180,E1 17122.278,E2 17122.278} C_VEL
LIN {X 0,Y 287.507,Z 781.698,A -85,B 0,C 180,E1 17127.749,E2 17127.749} C_VEL
LIN {X 0,Y 301.085,Z 806.25,A -85,B 0,C 180,E1 17133.791,E2 17133.791} C_VEL
LIN {X 0,Y 310.091,Z 829.214,A -85,B 0,C 180,E1 17138.048,E2 17138.048} C_VEL
LIN {X 0,Y 312.3,Z 847.496,A -85,B 0,C 180,E1 17140.435,E2 17140.435} C_VEL
LIN {X 0,Y 302.475,Z 882.339,A -85,B 0,C 180,E1 17143.201,E2 17143.201} C_VEL
LIN {X 0,Y 290.95,Z 914.604,A -85,B 0,C 180,E1 17147.128,E2 17147.128} C_VEL
LIN {X 0,Y 279.337,Z 942.867,A -85,B 0,C 180,E1 17152.195,E2 17152.195} C_VEL
LIN {X 0,Y 268.363,Z 967.757,A -85,B 0,C 180,E1 17158.759,E2 17158.759} C_VEL
LIN {X 0,Y 260.645,Z 986.311,A -85,B 0,C 180,E1 17166.006,E2 17166.006} C_VEL
LIN {X 0,Y 256.461,Z 999.372,A -85,B 0,C 180,E1 17173.714,E2 17173.714} C_VEL
LIN {X 0,Y 255.093,Z 1007.17,A -85,B 0,C 180,E1 17181.466,E2 17181.466} C_VEL
LIN {X 0,Y 254.942,Z 1009.647,A -85,B 0,C 180,E1 17186.595,E2 17186.595} C_VEL
LIN {X 0,Y 255.115,Z 1010.179,A -85,B 0,C 180,E1 17189.999,E2 17189.999} C_VEL
LIN {X 0,Y 255.046,Z 1008.24,A -85,B 0,C 180,E1 17196.818,E2 17196.818} C_VEL
LIN {X 0,Y 256.006,Z 1001.559,A -85,B 0,C 180,E1 17204.557,E2 17204.557} C_VEL
LIN {X 0,Y 260.091,Z 988.145,A -85,B 0,C 180,E1 17213.137,E2 17213.137} C_VEL
LIN {X 0,Y 267.588,Z 969.718,A -85,B 0,C 180,E1 17220.613,E2 17220.613} C_VEL
LIN {X 0,Y 278.001,Z 946.07,A -85,B 0,C 180,E1 17227.114,E2 17227.114} C_VEL
LIN {X 0,Y 290.038,Z 917.295,A -85,B 0,C 180,E1 17232.483,E2 17232.483} C_VEL
LIN {X 0,Y 303.298,Z 883.074,A -85,B 0,C 180,E1 17236.894,E2 17236.894} C_VEL
LIN {X 0,Y 319.799,Z 858.5,A -85,B 0,C 180,E1 17240.032,E2 17240.032} C_VEL
LIN {X 0,Y 320.584,Z 857.253,A -85,B 0,C 180,E1 17240.442,E2 17240.442} C_VEL
LIN {X 0,Y 302.14,Z 882.374,A -85,B 0,C 180,E1 17244.82,E2 17244.82} C_VEL
LIN {X 0,Y 287.516,Z 900.94,A -85,B 0,C 180,E1 17249.991,E2 17249.991} C_VEL
LIN {X 0,Y 279.216,Z 910.256,A -85,B 0,C 180,E1 17253.885,E2 17253.885} C_VEL
LIN {X 0,Y 270.382,Z 916.939,A -85,B 0,C 180,E1 17256.73,E2 17256.73} C_VEL
LIN {X 0,Y 262.772,Z 921.39,A -85,B 0,C 180,E1 17259.415,E2 17259.415} C_VEL
LIN {X 0,Y 262.113,Z 921.762,A -85,B 0,C 180,E1 17259.862,E2 17259.862} C_VEL
LIN {X 0,Y 255.516,Z 924.5,A -85,B 0,C 180,E1 17266.298,E2 17266.298} C_VEL
LIN {X 0,Y 251.826,Z 922.166,A -85,B 0,C 180,E1 17273.102,E2 17273.102} C_VEL
LIN {X 0,Y 250.419,Z 914.544,A -85,B 0,C 180,E1 17280.008,E2 17280.008} C_VEL
LIN {X 0,Y 251.123,Z 900.763,A -85,B 0,C 180,E1 17286.933,E2 17286.933} C_VEL
LIN {X 0,Y 253.37,Z 882.28,A -85,B 0,C 180,E1 17292.957,E2 17292.957} C_VEL
LIN {X 0,Y 256.614,Z 859.556,A -85,B 0,C 180,E1 17298.052,E2 17298.052} C_VEL
LIN {X 0,Y 260.371,Z 832.323,A -85,B 0,C 180,E1 17302.214,E2 17302.214} C_VEL
LIN {X 0,Y 261.326,Z 826.585,A -85,B 0,C 180,E1 17303.028,E2 17303.028} C_VEL
LIN {X 0,Y 264.74,Z 823.904,A -85,B 0,C 180,E1 17304.215,E2 17304.215} C_VEL
LIN {X 0,Y 272.248,Z 813.138,A -85,B 0,C 180,E1 17305.838,E2 17305.838} C_VEL
LIN {X 0,Y 280.224,Z 802.868,A -85,B 0,C 180,E1 17307.76,E2 17307.76} C_VEL
LIN {X 0,Y 287.084,Z 794.513,A -85,B 0,C 180,E1 17309.422,E2 17309.422} C_VEL
LIN {X 0,Y 296.799,Z 817.305,A -85,B 0,C 180,E1 17315.117,E2 17315.117} C_VEL
LIN {X 0,Y 303.511,Z 842.174,A -85,B 0,C 180,E1 17320.201,E2 17320.201} C_VEL
LIN {X 0,Y 303.885,Z 848.619,A -85,B 0,C 180,E1 17321.257,E2 17321.257} C_VEL
LIN {X 0,Y 292.618,Z 882.099,A -85,B 0,C 180,E1 17324.909,E2 17324.909} C_VEL
LIN {X 0,Y 280.478,Z 911.239,A -85,B 0,C 180,E1 17329.625,E2 17329.625} C_VEL
LIN {X 0,Y 268.529,Z 936.603,A -85,B 0,C 180,E1 17335.678,E2 17335.678} C_VEL
LIN {X 0,Y 258.329,Z 956.977,A -85,B 0,C 180,E1 17342.985,E2 17342.985} C_VEL
LIN {X 0,Y 251.763,Z 971.004,A -85,B 0,C 180,E1 17350.685,E2 17350.685} C_VEL
LIN {X 0,Y 248.066,Z 980.476,A -85,B 0,C 180,E1 17359.45,E2 17359.45} C_VEL
LIN {X 0,Y 247.06,Z 983.862,A -85,B 0,C 180,E1 17366.487,E2 17366.487} C_VEL
LIN {X 0,Y 247.131,Z 983.825,A -85,B 0,C 180,E1 17373.513,E2 17373.513} C_VEL
LIN {X 0,Y 248.431,Z 979.281,A -85,B 0,C 180,E1 17381.885,E2 17381.885} C_VEL
LIN {X 0,Y 252.371,Z 969.549,A -85,B 0,C 180,E1 17390.18,E2 17390.18} C_VEL
LIN {X 0,Y 260.025,Z 953.597,A -85,B 0,C 180,E1 17398.349,E2 17398.349} C_VEL
LIN {X 0,Y 270.252,Z 932.909,A -85,B 0,C 180,E1 17405.233,E2 17405.233} C_VEL
LIN {X 0,Y 282.407,Z 906.905,A -85,B 0,C 180,E1 17411.083,E2 17411.083} C_VEL
LIN {X 0,Y 294.712,Z 876.228,A -85,B 0,C 180,E1 17415.729,E2 17415.729} C_VEL
LIN {X 0,Y 304.103,Z 846.315,A -85,B 0,C 180,E1 17418.903,E2 17418.903} C_VEL
LIN {X 0,Y 298.159,Z 821.702,A -85,B 0,C 180,E1 17423.815,E2 17423.815} C_VEL
LIN {X 0,Y 288.938,Z 798.314,A -85,B 0,C 180,E1 17429.378,E2 17429.378} C_VEL
LIN {X 0,Y 278.798,Z 779.761,A -85,B 0,C 180,E1 17435.21,E2 17435.21} C_VEL
LIN {X 0,Y 271.542,Z 768.638,A -85,B 0,C 180,E1 17439.918,E2 17439.918} C_VEL
LIN {X 0,Y 267.5,Z 762.788,A -85,B 0,C 180,E1 17443.025,E2 17443.025} C_VEL
LIN {X 0,Y 263.161,Z 756.227,A -85,B 0,C 180,E1 17447.322,E2 17447.322} C_VEL
LIN {X 0,Y 259.322,Z 750.331,A -85,B 0,C 180,E1 17453.392,E2 17453.392} C_VEL
LIN {X 0,Y 258.291,Z 748.885,A -85,B 0,C 180,E1 17456.632,E2 17456.632} C_VEL
LIN {X 0,Y 259.319,Z 749.871,A -85,B 0,C 180,E1 17465.962,E2 17465.962} C_VEL
LIN {X 0,Y 262.688,Z 755.905,A -85,B 0,C 180,E1 17471.629,E2 17471.629} C_VEL
LIN {X 0,Y 264.544,Z 758.065,A -85,B 0,C 180,E1 17473.648,E2 17473.648} C_VEL
LIN {X 0,Y 269.934,Z 766.284,A -85,B 0,C 180,E1 17478.375,E2 17478.375} C_VEL
LIN {X 0,Y 277.583,Z 776.937,A -85,B 0,C 180,E1 17483.285,E2 17483.285} C_VEL
LIN {X 0,Y 290.142,Z 798.105,A -85,B 0,C 180,E1 17489.818,E2 17489.818} C_VEL
LIN {X 0,Y 301.32,Z 822.576,A -85,B 0,C 180,E1 17495.28,E2 17495.28} C_VEL
LIN {X 0,Y 305.188,Z 835.465,A -85,B 0,C 180,E1 17497.546,E2 17497.546} C_VEL
LIN {X 0,Y 306.799,Z 848.772,A -85,B 0,C 180,E1 17499.406,E2 17499.406} C_VEL
LIN {X 0,Y 296.507,Z 883.478,A -85,B 0,C 180,E1 17502.231,E2 17502.231} C_VEL
LIN {X 0,Y 284.538,Z 915.563,A -85,B 0,C 180,E1 17506.23,E2 17506.23} C_VEL
LIN {X 0,Y 272.461,Z 943.63,A -85,B 0,C 180,E1 17511.404,E2 17511.404} C_VEL
LIN {X 0,Y 261.378,Z 967.529,A -85,B 0,C 180,E1 17517.901,E2 17517.901} C_VEL
LIN {X 0,Y 253.25,Z 985.894,A -85,B 0,C 180,E1 17525.259,E2 17525.259} C_VEL
LIN {X 0,Y 248.72,Z 998.956,A -85,B 0,C 180,E1 17533.192,E2 17533.192} C_VEL
LIN {X 0,Y 247.213,Z 1006.759,A -85,B 0,C 180,E1 17541.192,E2 17541.192} C_VEL
LIN {X 0,Y 247.037,Z 1009.239,A -85,B 0,C 180,E1 17546.486,E2 17546.486} C_VEL
LIN {X 0,Y 247.219,Z 1009.772,A -85,B 0,C 180,E1 17549.999,E2 17549.999} C_VEL
LIN {X 0,Y 247.147,Z 1007.831,A -85,B 0,C 180,E1 17557.037,E2 17557.037} C_VEL
LIN {X 0,Y 248.203,Z 1001.144,A -85,B 0,C 180,E1 17565.026,E2 17565.026} C_VEL
LIN {X 0,Y 251.996,Z 989.341,A -85,B 0,C 180,E1 17572.988,E2 17572.988} C_VEL
LIN {X 0,Y 260.085,Z 970.529,A -85,B 0,C 180,E1 17581.108,E2 17581.108} C_VEL
LIN {X 0,Y 270.319,Z 948.305,A -85,B 0,C 180,E1 17587.526,E2 17587.526} C_VEL
LIN {X 0,Y 282.319,Z 921.298,A -85,B 0,C 180,E1 17592.877,E2 17592.877} C_VEL
LIN {X 0,Y 294.645,Z 892.034,A -85,B 0,C 180,E1 17597.076,E2 17597.076} C_VEL
LIN {X 0,Y 310.647,Z 870.773,A -85,B 0,C 180,E1 17600.204,E2 17600.204} C_VEL
LIN {X 0,Y 311.234,Z 869.887,A -85,B 0,C 180,E1 17600.605,E2 17600.605} C_VEL
LIN {X 0,Y 292.604,Z 892.119,A -85,B 0,C 180,E1 17605.316,E2 17605.316} C_VEL
LIN {X 0,Y 276.968,Z 909.084,A -85,B 0,C 180,E1 17611.136,E2 17611.136} C_VEL
LIN {X 0,Y 266.744,Z 918.418,A -85,B 0,C 180,E1 17616.598,E2 17616.598} C_VEL
LIN {X 0,Y 262.113,Z 921.762,A -85,B 0,C 180,E1 17619.862,E2 17619.862} C_VEL
LIN {X 0,Y 254.294,Z 924.89,A -85,B 0,C 180,E1 17623.271,E2 17623.271} C_VEL
LIN {X 0,Y 247.343,Z 926.105,A -85,B 0,C 180,E1 17626.772,E2 17626.772} C_VEL
LIN {X 0,Y 247.247,Z 925.959,A -85,B 0,C 180,E1 17626.896,E2 17626.896} C_VEL
LIN {X 0,Y 243.928,Z 923.116,A -85,B 0,C 180,E1 17633.28,E2 17633.28} C_VEL
LIN {X 0,Y 242.546,Z 913.859,A -85,B 0,C 180,E1 17640.95,E2 17640.95} C_VEL
LIN {X 0,Y 243.511,Z 898.878,A -85,B 0,C 180,E1 17648.05,E2 17648.05} C_VEL
LIN {X 0,Y 246.146,Z 878.869,A -85,B 0,C 180,E1 17654.251,E2 17654.251} C_VEL
LIN {X 0,Y 249.87,Z 854.161,A -85,B 0,C 180,E1 17659.482,E2 17659.482} C_VEL
LIN {X 0,Y 251.852,Z 842.113,A -85,B 0,C 180,E1 17661.613,E2 17661.613} C_VEL
LIN {X 0,Y 255.878,Z 838.994,A -85,B 0,C 180,E1 17663.087,E2 17663.087} C_VEL
LIN {X 0,Y 260.24,Z 833.561,A -85,B 0,C 180,E1 17664.04,E2 17664.04} C_VEL
LIN {X 0,Y 266.596,Z 827.303,A -85,B 0,C 180,E1 17665.83,E2 17665.83} C_VEL
LIN {X 0,Y 273.198,Z 818.316,A -85,B 0,C 180,E1 17667.124,E2 17667.124} C_VEL
LIN {X 0,Y 284.706,Z 804.418,A -85,B 0,C 180,E1 17669.67,E2 17669.67} C_VEL
LIN {X 0,Y 292.026,Z 822.338,A -85,B 0,C 180,E1 17674.373,E2 17674.373} C_VEL
LIN {X 0,Y 298.051,Z 847.138,A -85,B 0,C 180,E1 17679.663,E2 17679.663} C_VEL
LIN {X 0,Y 297.983,Z 851.536,A -85,B 0,C 180,E1 17680.345,E2 17680.345} C_VEL
LIN {X 0,Y 286.572,Z 883.727,A -85,B 0,C 180,E1 17683.957,E2 17683.957} C_VEL
LIN {X 0,Y 274.442,Z 911.639,A -85,B 0,C 180,E1 17688.545,E2 17688.545} C_VEL
LIN {X 0,Y 261.966,Z 937.008,A -85,B 0,C 180,E1 17694.693,E2 17694.693} C_VEL
LIN {X 0,Y 251.222,Z 957.385,A -85,B 0,C 180,E1 17702.155,E2 17702.155} C_VEL
LIN {X 0,Y 244.238,Z 971.414,A -85,B 0,C 180,E1 17710.065,E2 17710.065} C_VEL
LIN {X 0,Y 240.259,Z 980.884,A -85,B 0,C 180,E1 17719.103,E2 17719.103} C_VEL
LIN {X 0,Y 239.169,Z 984.269,A -85,B 0,C 180,E1 17726.371,E2 17726.371} C_VEL
LIN {X 0,Y 239.257,Z 984.232,A -85,B 0,C 180,E1 17733.629,E2 17733.629} C_VEL
LIN {X 0,Y 240.258,Z 980.806,A -85,B 0,C 180,E1 17740.898,E2 17740.898} C_VEL
LIN {X 0,Y 244.273,Z 971.25,A -85,B 0,C 180,E1 17749.933,E2 17749.933} C_VEL
LIN {X 0,Y 251.306,Z 957.142,A -85,B 0,C 180,E1 17757.836,E2 17757.836} C_VEL
LIN {X 0,Y 262.081,Z 936.679,A -85,B 0,C 180,E1 17765.291,E2 17765.291} C_VEL
LIN {X 0,Y 274.609,Z 911.168,A -85,B 0,C 180,E1 17771.425,E2 17771.425} C_VEL
LIN {X 0,Y 287.239,Z 881.883,A -85,B 0,C 180,E1 17776.179,E2 17776.179} C_VEL
LIN {X 0,Y 298.28,Z 849.352,A -85,B 0,C 180,E1 17779.799,E2 17779.799} C_VEL
LIN {X 0,Y 292.59,Z 824.498,A -85,B 0,C 180,E1 17785.007,E2 17785.007} C_VEL
LIN {X 0,Y 283.862,Z 801.678,A -85,B 0,C 180,E1 17790.813,E2 17790.813} C_VEL
LIN {X 0,Y 274.09,Z 782.96,A -85,B 0,C 180,E1 17797.138,E2 17797.138} C_VEL
LIN {X 0,Y 266.02,Z 770.383,A -85,B 0,C 180,E1 17803.353,E2 17803.353} C_VEL
LIN {X 0,Y 262.027,Z 763.999,A -85,B 0,C 180,E1 17807.478,E2 17807.478} C_VEL
LIN {X 0,Y 258.182,Z 758.009,A -85,B 0,C 180,E1 17813.785,E2 17813.785} C_VEL
LIN {X 0,Y 257.049,Z 756.562,A -85,B 0,C 180,E1 17818.305,E2 17818.305} C_VEL
LIN {X 0,Y 258.205,Z 757.767,A -85,B 0,C 180,E1 17825.671,E2 17825.671} C_VEL
LIN {X 0,Y 262.111,Z 764.033,A -85,B 0,C 180,E1 17832.079,E2 17832.079} C_VEL
LIN {X 0,Y 268.197,Z 773.597,A -85,B 0,C 180,E1 17837.868,E2 17837.868} C_VEL
LIN {X 0,Y 275.754,Z 784.967,A -85,B 0,C 180,E1 17843.021,E2 17843.021} C_VEL
LIN {X 0,Y 286.806,Z 804.655,A -85,B 0,C 180,E1 17849.221,E2 17849.221} C_VEL
LIN {X 0,Y 296.789,Z 828.047,A -85,B 0,C 180,E1 17854.624,E2 17854.624} C_VEL
LIN {X 0,Y 300.032,Z 840.354,A -85,B 0,C 180,E1 17856.851,E2 17856.851} C_VEL
LIN {X 0,Y 300.822,Z 851.914,A -85,B 0,C 180,E1 17858.468,E2 17858.468} C_VEL
LIN {X 0,Y 290.086,Z 886.157,A -85,B 0,C 180,E1 17861.383,E2 17861.383} C_VEL
LIN {X 0,Y 277.323,Z 918.608,A -85,B 0,C 180,E1 17865.611,E2 17865.611} C_VEL
LIN {X 0,Y 264.756,Z 946.165,A -85,B 0,C 180,E1 17871.018,E2 17871.018} C_VEL
LIN {X 0,Y 253.699,Z 968.807,A -85,B 0,C 180,E1 17877.511,E2 17877.511} C_VEL
LIN {X 0,Y 245.157,Z 987.256,A -85,B 0,C 180,E1 17885.362,E2 17885.362} C_VEL
LIN {X 0,Y 240.687,Z 999.702,A -85,B 0,C 180,E1 17893.555,E2 17893.555} C_VEL
LIN {X 0,Y 239.32,Z 1006.347,A -85,B 0,C 180,E1 17900.899,E2 17900.899} C_VEL
LIN {X 0,Y 239.132,Z 1008.831,A -85,B 0,C 180,E1 17906.369,E2 17906.369} C_VEL
LIN {X 0,Y 239.323,Z 1009.365,A -85,B 0,C 180,E1 17909.999,E2 17909.999} C_VEL
LIN {X 0,Y 239.28,Z 1007.423,A -85,B 0,C 180,E1 17917.27,E2 17917.27} C_VEL
LIN {X 0,Y 240.438,Z 1000.731,A -85,B 0,C 180,E1 17925.523,E2 17925.523} C_VEL
LIN {X 0,Y 244.552,Z 988.926,A -85,B 0,C 180,E1 17933.73,E2 17933.73} C_VEL
LIN {X 0,Y 253.136,Z 970.114,A -85,B 0,C 180,E1 17942.062,E2 17942.062} C_VEL
LIN {X 0,Y 263.944,Z 947.896,A -85,B 0,C 180,E1 17948.596,E2 17948.596} C_VEL
LIN {X 0,Y 276.934,Z 919.837,A -85,B 0,C 180,E1 17954.193,E2 17954.193} C_VEL
LIN {X 0,Y 285.11,Z 901.36,A -85,B 0,C 180,E1 17957.003,E2 17957.003} C_VEL
LIN {X 0,Y 301.363,Z 881.779,A -85,B 0,C 180,E1 17960.358,E2 17960.358} C_VEL
LIN {X 0,Y 301.937,Z 880.979,A -85,B 0,C 180,E1 17960.753,E2 17960.753} C_VEL
LIN {X 0,Y 282.923,Z 900.824,A -85,B 0,C 180,E1 17965.822,E2 17965.822} C_VEL
LIN {X 0,Y 267.484,Z 915.144,A -85,B 0,C 180,E1 17971.865,E2 17971.865} C_VEL
LIN {X 0,Y 255.17,Z 923.908,A -85,B 0,C 180,E1 17979.153,E2 17979.153} C_VEL
LIN {X 0,Y 248.023,Z 926.185,A -85,B 0,C 180,E1 17985.875,E2 17985.875} C_VEL
LIN {X 0,Y 247.247,Z 925.959,A -85,B 0,C 180,E1 17986.896,E2 17986.896} C_VEL
LIN {X 0,Y 241.058,Z 925.361,A -85,B 0,C 180,E1 17990.745,E2 17990.745} C_VEL
LIN {X 0,Y 235.606,Z 922.759,A -85,B 0,C 180,E1 17994.706,E2 17994.706} C_VEL
LIN {X 0,Y 234.686,Z 912.228,A -85,B 0,C 180,E1 18002.344,E2 18002.344} C_VEL
LIN {X 0,Y 235.951,Z 896.629,A -85,B 0,C 180,E1 18009.239,E2 18009.239} C_VEL
LIN {X 0,Y 238.72,Z 876.903,A -85,B 0,C 180,E1 18015.174,E2 18015.174} C_VEL
LIN {X 0,Y 242.119,Z 855.579,A -85,B 0,C 180,E1 18019.805,E2 18019.805} C_VEL
LIN {X 0,Y 246.395,Z 852.726,A -85,B 0,C 180,E1 18021.643,E2 18021.643} C_VEL
LIN {X 0,Y 249.977,Z 848.887,A -85,B 0,C 180,E1 18022.565,E2 18022.565} C_VEL
LIN {X 0,Y 256.007,Z 843.977,A -85,B 0,C 180,E1 18024.463,E2 18024.463} C_VEL
LIN {X 0,Y 269.04,Z 830.003,A -85,B 0,C 180,E1 18027.452,E2 18027.452} C_VEL
LIN {X 0,Y 281.441,Z 814.857,A -85,B 0,C 180,E1 18029.85,E2 18029.85} C_VEL
LIN {X 0,Y 282.634,Z 813.948,A -85,B 0,C 180,E1 18030.155,E2 18030.155} C_VEL
LIN {X 0,Y 289.661,Z 836.486,A -85,B 0,C 180,E1 18035.761,E2 18035.761} C_VEL
LIN {X 0,Y 292.306,Z 853.796,A -85,B 0,C 180,E1 18039.347,E2 18039.347} C_VEL
LIN {X 0,Y 280.523,Z 885.534,A -85,B 0,C 180,E1 18042.985,E2 18042.985} C_VEL
LIN {X 0,Y 267.628,Z 913.914,A -85,B 0,C 180,E1 18047.793,E2 18047.793} C_VEL
LIN {X 0,Y 254.759,Z 938.705,A -85,B 0,C 180,E1 18054.064,E2 18054.064} C_VEL
LIN {X 0,Y 244.18,Z 957.793,A -85,B 0,C 180,E1 18061.279,E2 18061.279} C_VEL
LIN {X 0,Y 236.736,Z 971.823,A -85,B 0,C 180,E1 18069.405,E2 18069.405} C_VEL
LIN {X 0,Y 232.458,Z 981.293,A -85,B 0,C 180,E1 18078.732,E2 18078.732} C_VEL
LIN {X 0,Y 231.279,Z 984.676,A -85,B 0,C 180,E1 18086.247,E2 18086.247} C_VEL
LIN {X 0,Y 231.365,Z 984.639,A -85,B 0,C 180,E1 18093.753,E2 18093.753} C_VEL
LIN {X 0,Y 232.954,Z 979.986,A -85,B 0,C 180,E1 18102.833,E2 18102.833} C_VEL
LIN {X 0,Y 237.429,Z 970.372,A -85,B 0,C 180,E1 18111.512,E2 18111.512} C_VEL
LIN {X 0,Y 245.943,Z 954.588,A -85,B 0,C 180,E1 18120.054,E2 18120.054} C_VEL
LIN {X 0,Y 257.033,Z 934.308,A -85,B 0,C 180,E1 18127.126,E2 18127.126} C_VEL
LIN {X 0,Y 269.841,Z 909.234,A -85,B 0,C 180,E1 18133.007,E2 18133.007} C_VEL
LIN {X 0,Y 282.821,Z 879.749,A -85,B 0,C 180,E1 18137.686,E2 18137.686} C_VEL
LIN {X 0,Y 292.38,Z 851.792,A -85,B 0,C 180,E1 18140.854,E2 18140.854} C_VEL
LIN {X 0,Y 287.299,Z 827.981,A -85,B 0,C 180,E1 18146.099,E2 18146.099} C_VEL
LIN {X 0,Y 278.998,Z 805.256,A -85,B 0,C 180,E1 18152.237,E2 18152.237} C_VEL
LIN {X 0,Y 270.849,Z 789.067,A -85,B 0,C 180,E1 18158.149,E2 18158.149} C_VEL
LIN {X 0,Y 264.154,Z 777.761,A -85,B 0,C 180,E1 18163.874,E2 18163.874} C_VEL
LIN {X 0,Y 260.309,Z 771.452,A -85,B 0,C 180,E1 18168.247,E2 18168.247} C_VEL
LIN {X 0,Y 256.869,Z 764.756,A -85,B 0,C 180,E1 18174.92,E2 18174.92} C_VEL
LIN {X 0,Y 257.055,Z 765.26,A -85,B 0,C 180,E1 18185.167,E2 18185.167} C_VEL
LIN {X 0,Y 260.792,Z 771.696,A -85,B 0,C 180,E1 18191.716,E2 18191.716} C_VEL
LIN {X 0,Y 266.938,Z 781.938,A -85,B 0,C 180,E1 18197.849,E2 18197.849} C_VEL
LIN {X 0,Y 273.354,Z 792.071,A -85,B 0,C 180,E1 18202.482,E2 18202.482} C_VEL
LIN {X 0,Y 283.321,Z 811.129,A -85,B 0,C 180,E1 18208.63,E2 18208.63} C_VEL
LIN {X 0,Y 292.164,Z 833.553,A -85,B 0,C 180,E1 18213.985,E2 18213.985} C_VEL
LIN {X 0,Y 294.84,Z 845.199,A -85,B 0,C 180,E1 18216.154,E2 18216.154} C_VEL
LIN {X 0,Y 295.094,Z 854.497,A -85,B 0,C 180,E1 18217.469,E2 18217.469} C_VEL
LIN {X 0,Y 283.605,Z 889.308,A -85,B 0,C 180,E1 18220.557,E2 18220.557} C_VEL
LIN {X 0,Y 270.136,Z 921.379,A -85,B 0,C 180,E1 18224.958,E2 18224.958} C_VEL
LIN {X 0,Y 257.688,Z 947.37,A -85,B 0,C 180,E1 18230.284,E2 18230.284} C_VEL
LIN {X 0,Y 245.641,Z 970.832,A -85,B 0,C 180,E1 18237.361,E2 18237.361} C_VEL
LIN {X 0,Y 237.071,Z 988.458,A -85,B 0,C 180,E1 18245.472,E2 18245.472} C_VEL
LIN {X 0,Y 232.67,Z 1000.288,A -85,B 0,C 180,E1 18253.944,E2 18253.944} C_VEL
LIN {X 0,Y 231.364,Z 1006.997,A -85,B 0,C 180,E1 18262.479,E2 18262.479} C_VEL
LIN {X 0,Y 231.426,Z 1008.959,A -85,B 0,C 180,E1 18269.999,E2 18269.999} C_VEL
LIN {X 0,Y 231.379,Z 1007.013,A -85,B 0,C 180,E1 18277.52,E2 18277.52} C_VEL
LIN {X 0,Y 232.709,Z 1000.319,A -85,B 0,C 180,E1 18286.052,E2 18286.052} C_VEL
LIN {X 0,Y 237.142,Z 988.511,A -85,B 0,C 180,E1 18294.519,E2 18294.519} C_VEL
LIN {X 0,Y 246.311,Z 969.702,A -85,B 0,C 180,E1 18303.062,E2 18303.062} C_VEL
LIN {X 0,Y 257.687,Z 947.489,A -85,B 0,C 180,E1 18309.715,E2 18309.715} C_VEL
LIN {X 0,Y 270.711,Z 920.492,A -85,B 0,C 180,E1 18315.203,E2 18315.203} C_VEL
LIN {X 0,Y 276.081,Z 909.174,A -85,B 0,C 180,E1 18317.035,E2 18317.035} C_VEL
LIN {X 0,Y 293.212,Z 890.355,A -85,B 0,C 180,E1 18320.766,E2 18320.766} C_VEL
LIN {X 0,Y 273.178,Z 908.556,A -85,B 0,C 180,E1 18326.351,E2 18326.351} C_VEL
LIN {X 0,Y 257.426,Z 920.794,A -85,B 0,C 180,E1 18332.892,E2 18332.892} C_VEL
LIN {X 0,Y 248.129,Z 926.161,A -85,B 0,C 180,E1 18338.533,E2 18338.533} C_VEL
LIN {X 0,Y 240.544,Z 927.831,A -85,B 0,C 180,E1 18345.426,E2 18345.426} C_VEL
LIN {X 0,Y 236.322,Z 924.616,A -85,B 0,C 180,E1 18352.647,E2 18352.647} C_VEL
LIN {X 0,Y 235.606,Z 922.759,A -85,B 0,C 180,E1 18354.706,E2 18354.706} C_VEL
LIN {X 0,Y 230.831,Z 918.386,A -85,B 0,C 180,E1 18358.704,E2 18358.704} C_VEL
LIN {X 0,Y 226.84,Z 912.196,A -85,B 0,C 180,E1 18362.719,E2 18362.719} C_VEL
LIN {X 0,Y 228.148,Z 896.769,A -85,B 0,C 180,E1 18369.558,E2 18369.558} C_VEL
LIN {X 0,Y 231.366,Z 874.636,A -85,B 0,C 180,E1 18376.156,E2 18376.156} C_VEL
LIN {X 0,Y 232.702,Z 867.653,A -85,B 0,C 180,E1 18378.01,E2 18378.01} C_VEL
LIN {X 0,Y 237.564,Z 864.29,A -85,B 0,C 180,E1 18380.201,E2 18380.201} C_VEL
LIN {X 0,Y 246.208,Z 857.462,A -85,B 0,C 180,E1 18383.146,E2 18383.146} C_VEL
LIN {X 0,Y 257.601,Z 847.304,A -85,B 0,C 180,E1 18386.161,E2 18386.161} C_VEL
LIN {X 0,Y 268.912,Z 836.062,A -85,B 0,C 180,E1 18388.6,E2 18388.6} C_VEL
LIN {X 0,Y 278.197,Z 825.201,A -85,B 0,C 180,E1 18390.235,E2 18390.235} C_VEL
LIN {X 0,Y 279.937,Z 824.188,A -85,B 0,C 180,E1 18390.7,E2 18390.7} C_VEL
LIN {X 0,Y 285.506,Z 846.257,A -85,B 0,C 180,E1 18396.193,E2 18396.193} C_VEL
LIN {X 0,Y 286.725,Z 856.056,A -85,B 0,C 180,E1 18398.312,E2 18398.312} C_VEL
LIN {X 0,Y 274.442,Z 887.606,A -85,B 0,C 180,E1 18402.007,E2 18402.007} C_VEL
LIN {X 0,Y 260.861,Z 916.12,A -85,B 0,C 180,E1 18407.001,E2 18407.001} C_VEL
LIN {X 0,Y 247.553,Z 940.404,A -85,B 0,C 180,E1 18413.393,E2 18413.393} C_VEL
LIN {X 0,Y 236.112,Z 960.091,A -85,B 0,C 180,E1 18421.253,E2 18421.253} C_VEL
LIN {X 0,Y 228.635,Z 973.493,A -85,B 0,C 180,E1 18429.656,E2 18429.656} C_VEL
LIN {X 0,Y 224.695,Z 981.7,A -85,B 0,C 180,E1 18438.338,E2 18438.338} C_VEL
LIN {X 0,Y 223.39,Z 985.083,A -85,B 0,C 180,E1 18446.114,E2 18446.114} C_VEL
LIN {X 0,Y 223.474,Z 985.047,A -85,B 0,C 180,E1 18453.885,E2 18453.885} C_VEL
LIN {X 0,Y 225.196,Z 980.396,A -85,B 0,C 180,E1 18463.283,E2 18463.283} C_VEL
LIN {X 0,Y 230.001,Z 970.785,A -85,B 0,C 180,E1 18472.243,E2 18472.243} C_VEL
LIN {X 0,Y 239.297,Z 954.538,A -85,B 0,C 180,E1 18481.211,E2 18481.211} C_VEL
LIN {X 0,Y 250.84,Z 934.475,A -85,B 0,C 180,E1 18488.299,E2 18488.299} C_VEL
LIN {X 0,Y 264.444,Z 908.92,A -85,B 0,C 180,E1 18494.327,E2 18494.327} C_VEL
LIN {X 0,Y 277.89,Z 879.261,A -85,B 0,C 180,E1 18499.009,E2 18499.009} C_VEL
LIN {X 0,Y 286.61,Z 854.957,A -85,B 0,C 180,E1 18501.781,E2 18501.781} C_VEL
LIN {X 0,Y 282.241,Z 832.054,A -85,B 0,C 180,E1 18507.095,E2 18507.095} C_VEL
LIN {X 0,Y 274.764,Z 810.293,A -85,B 0,C 180,E1 18513.307,E2 18513.307} C_VEL
LIN {X 0,Y 267.436,Z 794.737,A -85,B 0,C 180,E1 18519.271,E2 18519.271} C_VEL
LIN {X 0,Y 261.722,Z 784.605,A -85,B 0,C 180,E1 18524.796,E2 18524.796} C_VEL
LIN {X 0,Y 258.64,Z 778.946,A -85,B 0,C 180,E1 18528.812,E2 18528.812} C_VEL
LIN {X 0,Y 255.602,Z 772.528,A -85,B 0,C 180,E1 18535.746,E2 18535.746} C_VEL
LIN {X 0,Y 255.963,Z 773.069,A -85,B 0,C 180,E1 18544.87,E2 18544.87} C_VEL
LIN {X 0,Y 260.293,Z 781.291,A -85,B 0,C 180,E1 18552.591,E2 18552.591} C_VEL
LIN {X 0,Y 267.115,Z 792.346,A -85,B 0,C 180,E1 18559.12,E2 18559.12} C_VEL
LIN {X 0,Y 276.264,Z 810.033,A -85,B 0,C 180,E1 18565.777,E2 18565.777} C_VEL
LIN {X 0,Y 285.133,Z 831.624,A -85,B 0,C 180,E1 18571.662,E2 18571.662} C_VEL
LIN {X 0,Y 289.513,Z 847.938,A -85,B 0,C 180,E1 18575.109,E2 18575.109} C_VEL
LIN {X 0,Y 289.292,Z 857.579,A -85,B 0,C 180,E1 18576.461,E2 18576.461} C_VEL
LIN {X 0,Y 277.253,Z 891.861,A -85,B 0,C 180,E1 18579.638,E2 18579.638} C_VEL
LIN {X 0,Y 264.118,Z 921.804,A -85,B 0,C 180,E1 18583.868,E2 18583.868} C_VEL
LIN {X 0,Y 250.67,Z 948.576,A -85,B 0,C 180,E1 18589.509,E2 18589.509} C_VEL
LIN {X 0,Y 238.211,Z 971.536,A -85,B 0,C 180,E1 18596.755,E2 18596.755} C_VEL
LIN {X 0,Y 229.705,Z 988.04,A -85,B 0,C 180,E1 18604.63,E2 18604.63} C_VEL
LIN {X 0,Y 224.916,Z 999.872,A -85,B 0,C 180,E1 18613.375,E2 18613.375} C_VEL
LIN {X 0,Y 223.468,Z 1006.587,A -85,B 0,C 180,E1 18622.211,E2 18622.211} C_VEL
LIN {X 0,Y 223.528,Z 1008.552,A -85,B 0,C 180,E1 18629.999,E2 18629.999} C_VEL
LIN {X 0,Y 223.483,Z 1006.603,A -85,B 0,C 180,E1 18637.787,E2 18637.787} C_VEL
LIN {X 0,Y 224.976,Z 999.905,A -85,B 0,C 180,E1 18646.62,E2 18646.62} C_VEL
LIN {X 0,Y 230.59,Z 986.485,A -85,B 0,C 180,E1 18656.309,E2 18656.309} C_VEL
LIN {X 0,Y 240.172,Z 968.064,A -85,B 0,C 180,E1 18664.567,E2 18664.567} C_VEL
LIN {X 0,Y 252.341,Z 945.459,A -85,B 0,C 180,E1 18671.301,E2 18671.301} C_VEL
LIN {X 0,Y 268.975,Z 914.205,A -85,B 0,C 180,E1 18677.631,E2 18677.631} C_VEL
LIN {X 0,Y 282.523,Z 900.6,A -85,B 0,C 180,E1 18680.729,E2 18680.729} C_VEL
LIN {X 0,Y 283.177,Z 899.882,A -85,B 0,C 180,E1 18681.1,E2 18681.1} C_VEL
LIN {X 0,Y 263.343,Z 915.43,A -85,B 0,C 180,E1 18686.904,E2 18686.904} C_VEL
LIN {X 0,Y 249.301,Z 924.534,A -85,B 0,C 180,E1 18692.913,E2 18692.913} C_VEL
LIN {X 0,Y 241.099,Z 928.347,A -85,B 0,C 180,E1 18697.875,E2 18697.875} C_VEL
LIN {X 0,Y 233.084,Z 929.484,A -85,B 0,C 180,E1 18704.949,E2 18704.949} C_VEL
LIN {X 0,Y 228.565,Z 925.734,A -85,B 0,C 180,E1 18712.396,E2 18712.396} C_VEL
LIN {X 0,Y 226.868,Z 916.796,A -85,B 0,C 180,E1 18720.009,E2 18720.009} C_VEL
LIN {X 0,Y 226.84,Z 912.196,A -85,B 0,C 180,E1 18722.719,E2 18722.719} C_VEL
LIN {X 0,Y 224.732,Z 906.517,A -85,B 0,C 180,E1 18725.67,E2 18725.67} C_VEL
LIN {X 0,Y 220.535,Z 896.546,A -85,B 0,C 180,E1 18729.965,E2 18729.965} C_VEL
LIN {X 0,Y 220.588,Z 895.262,A -85,B 0,C 180,E1 18730.434,E2 18730.434} C_VEL
LIN {X 0,Y 223.168,Z 878.559,A -85,B 0,C 180,E1 18735.755,E2 18735.755} C_VEL
LIN {X 0,Y 228.178,Z 875.298,A -85,B 0,C 180,E1 18738.38,E2 18738.38} C_VEL
LIN {X 0,Y 243.247,Z 864.635,A -85,B 0,C 180,E1 18743.951,E2 18743.951} C_VEL
LIN {X 0,Y 257.878,Z 852.12,A -85,B 0,C 180,E1 18747.547,E2 18747.547} C_VEL
LIN {X 0,Y 270.41,Z 840.111,A -85,B 0,C 180,E1 18750.017,E2 18750.017} C_VEL
LIN {X 0,Y 276.235,Z 833.528,A -85,B 0,C 180,E1 18750.928,E2 18750.928} C_VEL
LIN {X 0,Y 280.289,Z 851.38,A -85,B 0,C 180,E1 18755.582,E2 18755.582} C_VEL
LIN {X 0,Y 280.584,Z 860.1,A -85,B 0,C 180,E1 18757.4,E2 18757.4} C_VEL
LIN {X 0,Y 266.902,Z 892.994,A -85,B 0,C 180,E1 18761.496,E2 18761.496} C_VEL
LIN {X 0,Y 253.194,Z 919.945,A -85,B 0,C 180,E1 18766.553,E2 18766.553} C_VEL
LIN {X 0,Y 239.615,Z 943.396,A -85,B 0,C 180,E1 18773.11,E2 18773.11} C_VEL
LIN {X 0,Y 228.015,Z 962.249,A -85,B 0,C 180,E1 18781.222,E2 18781.222} C_VEL
LIN {X 0,Y 220.487,Z 975.008,A -85,B 0,C 180,E1 18789.919,E2 18789.919} C_VEL
LIN {X 0,Y 216.403,Z 983.262,A -85,B 0,C 180,E1 18799.927,E2 18799.927} C_VEL
LIN {X 0,Y 215.591,Z 985.935,A -85,B 0,C 180,E1 18810.001,E2 18810.001} C_VEL
LIN {X 0,Y 216.408,Z 983.186,A -85,B 0,C 180,E1 18820.074,E2 18820.074} C_VEL
LIN {X 0,Y 220.52,Z 974.874,A -85,B 0,C 180,E1 18830.079,E2 18830.079} C_VEL
LIN {X 0,Y 228.101,Z 962.041,A -85,B 0,C 180,E1 18838.767,E2 18838.767} C_VEL
LIN {X 0,Y 239.728,Z 943.082,A -85,B 0,C 180,E1 18846.871,E2 18846.871} C_VEL
LIN {X 0,Y 253.322,Z 919.534,A -85,B 0,C 180,E1 18853.421,E2 18853.421} C_VEL
LIN {X 0,Y 267.182,Z 892.28,A -85,B 0,C 180,E1 18858.486,E2 18858.486} C_VEL
LIN {X 0,Y 280.551,Z 859.789,A -85,B 0,C 180,E1 18862.521,E2 18862.521} C_VEL
LIN {X 0,Y 278.892,Z 844.275,A -85,B 0,C 180,E1 18866.034,E2 18866.034} C_VEL
LIN {X 0,Y 273.316,Z 822.829,A -85,B 0,C 180,E1 18871.904,E2 18871.904} C_VEL
LIN {X 0,Y 266.083,Z 804.351,A -85,B 0,C 180,E1 18878.517,E2 18878.517} C_VEL
LIN {X 0,Y 259.794,Z 792.115,A -85,B 0,C 180,E1 18885.113,E2 18885.113} C_VEL
LIN {X 0,Y 256.933,Z 786.54,A -85,B 0,C 180,E1 18889.166,E2 18889.166} C_VEL
LIN {X 0,Y 254.415,Z 780.338,A -85,B 0,C 180,E1 18895.726,E2 18895.726} C_VEL
LIN {X 0,Y 254.703,Z 781.003,A -85,B 0,C 180,E1 18904.681,E2 18904.681} C_VEL
LIN {X 0,Y 258.588,Z 788.74,A -85,B 0,C 180,E1 18912.139,E2 18912.139} C_VEL
LIN {X 0,Y 264.901,Z 799.932,A -85,B 0,C 180,E1 18918.745,E2 18918.745} C_VEL
LIN {X 0,Y 272.975,Z 816.842,A -85,B 0,C 180,E1 18925.262,E2 18925.262} C_VEL
LIN {X 0,Y 280.837,Z 837.707,A -85,B 0,C 180,E1 18931.103,E2 18931.103} C_VEL
LIN {X 0,Y 284.25,Z 852.579,A -85,B 0,C 180,E1 18934.361,E2 18934.361} C_VEL
LIN {X 0,Y 283.802,Z 859.792,A -85,B 0,C 180,E1 18935.361,E2 18935.361} C_VEL
LIN {X 0,Y 271.263,Z 893.72,A -85,B 0,C 180,E1 18938.607,E2 18938.607} C_VEL
LIN {X 0,Y 257.206,Z 924.179,A -85,B 0,C 180,E1 18943.061,E2 18943.061} C_VEL
LIN {X 0,Y 242.636,Z 951.555,A -85,B 0,C 180,E1 18949.18,E2 18949.18} C_VEL
LIN {X 0,Y 230.2,Z 973.335,A -85,B 0,C 180,E1 18956.574,E2 18956.574} C_VEL
LIN {X 0,Y 220.858,Z 990.771,A -85,B 0,C 180,E1 18965.711,E2 18965.711} C_VEL
LIN {X 0,Y 216.343,Z 1002.244,A -85,B 0,C 180,E1 18975.82,E2 18975.82} C_VEL
LIN {X 0,Y 215.578,Z 1006.176,A -85,B 0,C 180,E1 18981.924,E2 18981.924} C_VEL
LIN {X 0,Y 215.63,Z 1008.145,A -85,B 0,C 180,E1 18989.999,E2 18989.999} C_VEL
LIN {X 0,Y 215.593,Z 1006.194,A -85,B 0,C 180,E1 18998.074,E2 18998.074} C_VEL
LIN {X 0,Y 217.237,Z 999.49,A -85,B 0,C 180,E1 19007.23,E2 19007.23} C_VEL
LIN {X 0,Y 223.325,Z 986.069,A -85,B 0,C 180,E1 19017.234,E2 19017.234} C_VEL
LIN {X 0,Y 233.493,Z 967.648,A -85,B 0,C 180,E1 19025.704,E2 19025.704} C_VEL
LIN {X 0,Y 246.323,Z 945.051,A -85,B 0,C 180,E1 19032.543,E2 19032.543} C_VEL
LIN {X 0,Y 259.34,Z 921.226,A -85,B 0,C 180,E1 19037.586,E2 19037.586} C_VEL
LIN {X 0,Y 273.08,Z 908.572,A -85,B 0,C 180,E1 19040.916,E2 19040.916} C_VEL
LIN {X 0,Y 268.346,Z 911.709,A -85,B 0,C 180,E1 19042.671,E2 19042.671} C_VEL
LIN {X 0,Y 249.635,Z 923.672,A -85,B 0,C 180,E1 19048.977,E2 19048.977} C_VEL
LIN {X 0,Y 239.613,Z 928.613,A -85,B 0,C 180,E1 19053.758,E2 19053.758} C_VEL
LIN {X 0,Y 229.451,Z 931.389,A -85,B 0,C 180,E1 19060.745,E2 19060.745} C_VEL
LIN {X 0,Y 222.816,Z 929.559,A -85,B 0,C 180,E1 19068.247,E2 19068.247} C_VEL
LIN {X 0,Y 219.536,Z 922.821,A -85,B 0,C 180,E1 19076.054,E2 19076.054} C_VEL
LIN {X 0,Y 219.109,Z 910.473,A -85,B 0,C 180,E1 19083.971,E2 19083.971} C_VEL
LIN {X 0,Y 220.588,Z 895.262,A -85,B 0,C 180,E1 19090.434,E2 19090.434} C_VEL
LIN {X 0,Y 220.187,Z 887.771,A -85,B 0,C 180,E1 19094.544,E2 19094.544} C_VEL
LIN {X 0,Y 222.514,Z 883.279,A -85,B 0,C 180,E1 19098.246,E2 19098.246} C_VEL
LIN {X 0,Y 223.442,Z 882.612,A -85,B 0,C 180,E1 19098.718,E2 19098.718} C_VEL
LIN {X 0,Y 241.26,Z 870.62,A -85,B 0,C 180,E1 19105.07,E2 19105.07} C_VEL
LIN {X 0,Y 256.575,Z 858.431,A -85,B 0,C 180,E1 19108.665,E2 19108.665} C_VEL
LIN {X 0,Y 271.251,Z 844.978,A -85,B 0,C 180,E1 19111.32,E2 19111.32} C_VEL
LIN {X 0,Y 272.71,Z 843.356,A -85,B 0,C 180,E1 19111.507,E2 19111.507} C_VEL
LIN {X 0,Y 275.436,Z 861.631,A -85,B 0,C 180,E1 19116.206,E2 19116.206} C_VEL
LIN {X 0,Y 261.594,Z 893.606,A -85,B 0,C 180,E1 19120.226,E2 19120.226} C_VEL
LIN {X 0,Y 247.063,Z 921.053,A -85,B 0,C 180,E1 19125.445,E2 19125.445} C_VEL
LIN {X 0,Y 232.468,Z 945.057,A -85,B 0,C 180,E1 19132.367,E2 19132.367} C_VEL
LIN {X 0,Y 221.018,Z 962.665,A -85,B 0,C 180,E1 19140.226,E2 19140.226} C_VEL
LIN {X 0,Y 213.012,Z 975.417,A -85,B 0,C 180,E1 19149.183,E2 19149.183} C_VEL
LIN {X 0,Y 208.567,Z 983.762,A -85,B 0,C 180,E1 19159.715,E2 19159.715} C_VEL
LIN {X 0,Y 207.697,Z 986.342,A -85,B 0,C 180,E1 19170.001,E2 19170.001} C_VEL
LIN {X 0,Y 208.571,Z 983.689,A -85,B 0,C 180,E1 19180.284,E2 19180.284} C_VEL
LIN {X 0,Y 213.046,Z 975.285,A -85,B 0,C 180,E1 19190.815,E2 19190.815} C_VEL
LIN {X 0,Y 221.131,Z 962.452,A -85,B 0,C 180,E1 19199.764,E2 19199.764} C_VEL
LIN {X 0,Y 233.371,Z 943.493,A -85,B 0,C 180,E1 19208.051,E2 19208.051} C_VEL
LIN {X 0,Y 247.439,Z 920.213,A -85,B 0,C 180,E1 19214.627,E2 19214.627} C_VEL
LIN {X 0,Y 261.889,Z 892.86,A -85,B 0,C 180,E1 19219.762,E2 19219.762} C_VEL
LIN {X 0,Y 275.269,Z 860.96,A -85,B 0,C 180,E1 19223.828,E2 19223.828} C_VEL
LIN {X 0,Y 271.916,Z 839.312,A -85,B 0,C 180,E1 19229.391,E2 19229.391} C_VEL
LIN {X 0,Y 266.138,Z 819.501,A -85,B 0,C 180,E1 19235.722,E2 19235.722} C_VEL
LIN {X 0,Y 260.052,Z 804.703,A -85,B 0,C 180,E1 19242.304,E2 19242.304} C_VEL
LIN {X 0,Y 255.217,Z 794.198,A -85,B 0,C 180,E1 19249.309,E2 19249.309} C_VEL
LIN {X 0,Y 252.818,Z 787.937,A -85,B 0,C 180,E1 19256.559,E2 19256.559} C_VEL
LIN {X 0,Y 253.255,Z 788.894,A -85,B 0,C 180,E1 19264.493,E2 19264.493} C_VEL
LIN {X 0,Y 256.772,Z 796.531,A -85,B 0,C 180,E1 19271.902,E2 19271.902} C_VEL
LIN {X 0,Y 262.291,Z 807.187,A -85,B 0,C 180,E1 19278.285,E2 19278.285} C_VEL
LIN {X 0,Y 269.779,Z 823.982,A -85,B 0,C 180,E1 19284.89,E2 19284.89} C_VEL
LIN {X 0,Y 276.826,Z 845.472,A -85,B 0,C 180,E1 19290.972,E2 19290.972} C_VEL
LIN {X 0,Y 279.017,Z 857.013,A -85,B 0,C 180,E1 19293.551,E2 19293.551} C_VEL
LIN {X 0,Y 277.69,Z 864.032,A -85,B 0,C 180,E1 19294.396,E2 19294.396} C_VEL
LIN {X 0,Y 264.551,Z 897.503,A -85,B 0,C 180,E1 19297.765,E2 19297.765} C_VEL
LIN {X 0,Y 249.709,Z 927.672,A -85,B 0,C 180,E1 19302.451,E2 19302.451} C_VEL
LIN {X 0,Y 235.509,Z 952.892,A -85,B 0,C 180,E1 19308.399,E2 19308.399} C_VEL
LIN {X 0,Y 222.752,Z 974.132,A -85,B 0,C 180,E1 19315.947,E2 19315.947} C_VEL
LIN {X 0,Y 213.485,Z 990.353,A -85,B 0,C 180,E1 19324.815,E2 19324.815} C_VEL
LIN {X 0,Y 208.545,Z 1001.829,A -85,B 0,C 180,E1 19335.279,E2 19335.279} C_VEL
LIN {X 0,Y 207.697,Z 1005.766,A -85,B 0,C 180,E1 19341.616,E2 19341.616} C_VEL
LIN {X 0,Y 207.731,Z 1007.738,A -85,B 0,C 180,E1 19349.999,E2 19349.999} C_VEL
LIN {X 0,Y 207.71,Z 1005.784,A -85,B 0,C 180,E1 19358.382,E2 19358.382} C_VEL
LIN {X 0,Y 209.533,Z 999.075,A -85,B 0,C 180,E1 19367.884,E2 19367.884} C_VEL
LIN {X 0,Y 216.123,Z 985.653,A -85,B 0,C 180,E1 19378.221,E2 19378.221} C_VEL
LIN {X 0,Y 226.966,Z 967.236,A -85,B 0,C 180,E1 19386.897,E2 19386.897} C_VEL
LIN {X 0,Y 240.424,Z 944.643,A -85,B 0,C 180,E1 19393.846,E2 19393.846} C_VEL
LIN {X 0,Y 251.522,Z 925.893,A -85,B 0,C 180,E1 19398.068,E2 19398.068} C_VEL
LIN {X 0,Y 264.266,Z 915.098,A -85,B 0,C 180,E1 19401.414,E2 19401.414} C_VEL
LIN {X 0,Y 243.43,Z 926.737,A -85,B 0,C 180,E1 19408.095,E2 19408.095} C_VEL
LIN {X 0,Y 232.93,Z 931.138,A -85,B 0,C 180,E1 19412.945,E2 19412.945} C_VEL
LIN {X 0,Y 222.216,Z 933.209,A -85,B 0,C 180,E1 19420.092,E2 19420.092} C_VEL
LIN {X 0,Y 215.184,Z 930.859,A -85,B 0,C 180,E1 19427.824,E2 19427.824} C_VEL
LIN {X 0,Y 211.712,Z 923.596,A -85,B 0,C 180,E1 19435.908,E2 19435.908} C_VEL
LIN {X 0,Y 211.246,Z 910.798,A -85,B 0,C 180,E1 19444.119,E2 19444.119} C_VEL
LIN {X 0,Y 213.199,Z 892.343,A -85,B 0,C 180,E1 19451.79,E2 19451.79} C_VEL
LIN {X 0,Y 213.946,Z 888.599,A -85,B 0,C 180,E1 19453.306,E2 19453.306} C_VEL
LIN {X 0,Y 223.442,Z 882.612,A -85,B 0,C 180,E1 19458.718,E2 19458.718} C_VEL
LIN {X 0,Y 227.711,Z 881.725,A -85,B 0,C 180,E1 19461.522,E2 19461.522} C_VEL
LIN {X 0,Y 232.553,Z 880.728,A -85,B 0,C 180,E1 19464.197,E2 19464.197} C_VEL
LIN {X 0,Y 243.214,Z 873.563,A -85,B 0,C 180,E1 19467.142,E2 19467.142} C_VEL
LIN {X 0,Y 256.987,Z 863.076,A -85,B 0,C 180,E1 19470.089,E2 19470.089} C_VEL
LIN {X 0,Y 267.941,Z 853.985,A -85,B 0,C 180,E1 19472.046,E2 19472.046} C_VEL
LIN {X 0,Y 268.95,Z 854.81,A -85,B 0,C 180,E1 19472.602,E2 19472.602} C_VEL
LIN {X 0,Y 269.586,Z 865.09,A -85,B 0,C 180,E1 19475.173,E2 19475.173} C_VEL
LIN {X 0,Y 255.525,Z 895.995,A -85,B 0,C 180,E1 19479.187,E2 19479.187} C_VEL
LIN {X 0,Y 240.305,Z 923.405,A -85,B 0,C 180,E1 19484.573,E2 19484.573} C_VEL
LIN {X 0,Y 225.198,Z 946.857,A -85,B 0,C 180,E1 19491.661,E2 19491.661} C_VEL
LIN {X 0,Y 212.922,Z 964.749,A -85,B 0,C 180,E1 19500.148,E2 19500.148} C_VEL
LIN {X 0,Y 204.253,Z 977.995,A -85,B 0,C 180,E1 19510.515,E2 19510.515} C_VEL
LIN {X 0,Y 200.302,Z 985.026,A -85,B 0,C 180,E1 19521.305,E2 19521.305} C_VEL
LIN {X 0,Y 199.802,Z 986.749,A -85,B 0,C 180,E1 19530.001,E2 19530.001} C_VEL
LIN {X 0,Y 200.317,Z 984.974,A -85,B 0,C 180,E1 19538.695,E2 19538.695} C_VEL
LIN {X 0,Y 204.278,Z 977.885,A -85,B 0,C 180,E1 19549.484,E2 19549.484} C_VEL
LIN {X 0,Y 213.031,Z 964.546,A -85,B 0,C 180,E1 19559.837,E2 19559.837} C_VEL
LIN {X 0,Y 225.385,Z 946.49,A -85,B 0,C 180,E1 19568.349,E2 19568.349} C_VEL
LIN {X 0,Y 240.617,Z 922.668,A -85,B 0,C 180,E1 19575.48,E2 19575.48} C_VEL
LIN {X 0,Y 255.748,Z 895.379,A -85,B 0,C 180,E1 19580.781,E2 19580.781} C_VEL
LIN {X 0,Y 269.653,Z 864.55,A -85,B 0,C 180,E1 19584.776,E2 19584.776} C_VEL
LIN {X 0,Y 266.922,Z 843.148,A -85,B 0,C 180,E1 19590.563,E2 19590.563} C_VEL
LIN {X 0,Y 262.122,Z 824.931,A -85,B 0,C 180,E1 19596.707,E2 19596.707} C_VEL
LIN {X 0,Y 256.881,Z 811.062,A -85,B 0,C 180,E1 19603.217,E2 19603.217} C_VEL
LIN {X 0,Y 252.826,Z 801.442,A -85,B 0,C 180,E1 19610.078,E2 19610.078} C_VEL
LIN {X 0,Y 251.246,Z 795.657,A -85,B 0,C 180,E1 19616.538,E2 19616.538} C_VEL
LIN {X 0,Y 251.615,Z 796.536,A -85,B 0,C 180,E1 19624.198,E2 19624.198} C_VEL
LIN {X 0,Y 254.634,Z 804.074,A -85,B 0,C 180,E1 19631.568,E2 19631.568} C_VEL
LIN {X 0,Y 259.617,Z 814.44,A -85,B 0,C 180,E1 19637.886,E2 19637.886} C_VEL
LIN {X 0,Y 265.745,Z 829.597,A -85,B 0,C 180,E1 19644.031,E2 19644.031} C_VEL
LIN {X 0,Y 271.879,Z 849.965,A -85,B 0,C 180,E1 19650.07,E2 19650.07} C_VEL
LIN {X 0,Y 273.69,Z 861.373,A -85,B 0,C 180,E1 19652.725,E2 19652.725} C_VEL
LIN {X 0,Y 260.936,Z 894.309,A -85,B 0,C 180,E1 19656.027,E2 19656.027} C_VEL
LIN {X 0,Y 245.423,Z 925.352,A -85,B 0,C 180,E1 19660.682,E2 19660.682} C_VEL
LIN {X 0,Y 229.71,Z 952.199,A -85,B 0,C 180,E1 19666.98,E2 19666.98} C_VEL
LIN {X 0,Y 215.945,Z 973.883,A -85,B 0,C 180,E1 19674.812,E2 19674.812} C_VEL
LIN {X 0,Y 206.166,Z 989.935,A -85,B 0,C 180,E1 19683.854,E2 19683.854} C_VEL
LIN {X 0,Y 200.763,Z 1001.414,A -85,B 0,C 180,E1 19694.694,E2 19694.694} C_VEL
LIN {X 0,Y 199.803,Z 1005.355,A -85,B 0,C 180,E1 19701.282,E2 19701.282} C_VEL
LIN {X 0,Y 199.831,Z 1007.331,A -85,B 0,C 180,E1 19709.999,E2 19709.999} C_VEL
LIN {X 0,Y 199.902,Z 1004.764,A -85,B 0,C 180,E1 19720.128,E2 19720.128} C_VEL
LIN {X 0,Y 202.813,Z 996.562,A -85,B 0,C 180,E1 19730.711,E2 19730.711} C_VEL
LIN {X 0,Y 210.053,Z 983.459,A -85,B 0,C 180,E1 19740.302,E2 19740.302} C_VEL
LIN {X 0,Y 222.067,Z 964.374,A -85,B 0,C 180,E1 19749.1,E2 19749.1} C_VEL
LIN {X 0,Y 237.673,Z 939.191,A -85,B 0,C 180,E1 19756.438,E2 19756.438} C_VEL
LIN {X 0,Y 243.003,Z 930.677,A -85,B 0,C 180,E1 19758.39,E2 19758.39} C_VEL
LIN {X 0,Y 253.086,Z 922.85,A -85,B 0,C 180,E1 19761.052,E2 19761.052} C_VEL
LIN {X 0,Y 253.935,Z 921.97,A -85,B 0,C 180,E1 19761.764,E2 19761.764} C_VEL
LIN {X 0,Y 233.392,Z 931.307,A -85,B 0,C 180,E1 19768.747,E2 19768.747} C_VEL
LIN {X 0,Y 220.182,Z 934.807,A -85,B 0,C 180,E1 19775.643,E2 19775.643} C_VEL
LIN {X 0,Y 210.772,Z 934.149,A -85,B 0,C 180,E1 19783.312,E2 19783.312} C_VEL
LIN {X 0,Y 204.846,Z 927.841,A -85,B 0,C 180,E1 19792.578,E2 19792.578} C_VEL
LIN {X 0,Y 203.22,Z 916.719,A -85,B 0,C 180,E1 19801.077,E2 19801.077} C_VEL
LIN {X 0,Y 204.306,Z 900.504,A -85,B 0,C 180,E1 19809.07,E2 19809.07} C_VEL
LIN {X 0,Y 204.612,Z 898.177,A -85,B 0,C 180,E1 19810.131,E2 19810.131} C_VEL
LIN {X 0,Y 213.439,Z 892.731,A -85,B 0,C 180,E1 19816.493,E2 19816.493} C_VEL
LIN {X 0,Y 229.557,Z 882.861,A -85,B 0,C 180,E1 19823.32,E2 19823.32} C_VEL
LIN {X 0,Y 232.553,Z 880.728,A -85,B 0,C 180,E1 19824.197,E2 19824.197} C_VEL
LIN {X 0,Y 244.499,Z 877.197,A -85,B 0,C 180,E1 19829.041,E2 19829.041} C_VEL
LIN {X 0,Y 261.886,Z 864.373,A -85,B 0,C 180,E1 19832.336,E2 19832.336} C_VEL
LIN {X 0,Y 264.087,Z 863.888,A -85,B 0,C 180,E1 19833.008,E2 19833.008} C_VEL
LIN {X 0,Y 263.822,Z 868.484,A -85,B 0,C 180,E1 19834.095,E2 19834.095} C_VEL
LIN {X 0,Y 248.686,Z 900.097,A -85,B 0,C 180,E1 19838.384,E2 19838.384} C_VEL
LIN {X 0,Y 233.005,Z 926.619,A -85,B 0,C 180,E1 19843.907,E2 19843.907} C_VEL
LIN {X 0,Y 217.456,Z 949.383,A -85,B 0,C 180,E1 19851.198,E2 19851.198} C_VEL
LIN {X 0,Y 204.825,Z 966.839,A -85,B 0,C 180,E1 19860.069,E2 19860.069} C_VEL
LIN {X 0,Y 196.742,Z 978.405,A -85,B 0,C 180,E1 19869.739,E2 19869.739} C_VEL
LIN {X 0,Y 192.484,Z 985.434,A -85,B 0,C 180,E1 19880.949,E2 19880.949} C_VEL
LIN {X 0,Y 191.938,Z 987.154,A -85,B 0,C 180,E1 19890.001,E2 19890.001} C_VEL
LIN {X 0,Y 192.498,Z 985.381,A -85,B 0,C 180,E1 19899.051,E2 19899.051} C_VEL
LIN {X 0,Y 196.768,Z 978.296,A -85,B 0,C 180,E1 19910.26,E2 19910.26} C_VEL
LIN {X 0,Y 206.12,Z 964.958,A -85,B 0,C 180,E1 19920.945,E2 19920.945} C_VEL
LIN {X 0,Y 218.957,Z 947.176,A -85,B 0,C 180,E1 19929.542,E2 19929.542} C_VEL
LIN {X 0,Y 234.735,Z 923.681,A -85,B 0,C 180,E1 19936.72,E2 19936.72} C_VEL
LIN {X 0,Y 250.746,Z 895.877,A -85,B 0,C 180,E1 19942.174,E2 19942.174} C_VEL
LIN {X 0,Y 264.053,Z 866.766,A -85,B 0,C 180,E1 19946.095,E2 19946.095} C_VEL
LIN {X 0,Y 261.801,Z 846.415,A -85,B 0,C 180,E1 19951.945,E2 19951.945} C_VEL
LIN {X 0,Y 257.816,Z 829.589,A -85,B 0,C 180,E1 19958.002,E2 19958.002} C_VEL
LIN {X 0,Y 253.224,Z 815.786,A -85,B 0,C 180,E1 19965.011,E2 19965.011} C_VEL
LIN {X 0,Y 250.424,Z 808.725,A -85,B 0,C 180,E1 19970.641,E2 19970.641} C_VEL
LIN {X 0,Y 249.363,Z 803.325,A -85,B 0,C 180,E1 19976.511,E2 19976.511} C_VEL
LIN {X 0,Y 249.642,Z 804.136,A -85,B 0,C 180,E1 19983.904,E2 19983.904} C_VEL
LIN {X 0,Y 252.352,Z 811.491,A -85,B 0,C 180,E1 19991.236,E2 19991.236} C_VEL
LIN {X 0,Y 256.939,Z 822.116,A -85,B 0,C 180,E1 19997.697,E2 19997.697} C_VEL
LIN {X 0,Y 262.314,Z 837.076,A -85,B 0,C 180,E1 20003.822,E2 20003.822} C_VEL
LIN {X 0,Y 267.555,Z 857.616,A -85,B 0,C 180,E1 20009.969,E2 20009.969} C_VEL
LIN {X 0,Y 268.352,Z 865.046,A -85,B 0,C 180,E1 20011.733,E2 20011.733} C_VEL
LIN {X 0,Y 253.774,Z 899.314,A -85,B 0,C 180,E1 20015.25,E2 20015.25} C_VEL
LIN {X 0,Y 237.589,Z 929.464,A -85,B 0,C 180,E1 20020.116,E2 20020.116} C_VEL
LIN {X 0,Y 221.178,Z 955.91,A -85,B 0,C 180,E1 20026.798,E2 20026.798} C_VEL
LIN {X 0,Y 206.742,Z 977.327,A -85,B 0,C 180,E1 20035.418,E2 20035.418} C_VEL
LIN {X 0,Y 197.267,Z 992.294,A -85,B 0,C 180,E1 20045.029,E2 20045.029} C_VEL
LIN {X 0,Y 192.481,Z 1002.603,A -85,B 0,C 180,E1 20056.35,E2 20056.35} C_VEL
LIN {X 0,Y 191.693,Z 1006.38,A -85,B 0,C 180,E1 20065.469,E2 20065.469} C_VEL
LIN {X 0,Y 191.957,Z 1006.926,A -85,B 0,C 180,E1 20069.999,E2 20069.999} C_VEL
LIN {X 0,Y 192.028,Z 1004.352,A -85,B 0,C 180,E1 20080.548,E2 20080.548} C_VEL
LIN {X 0,Y 195.247,Z 996.187,A -85,B 0,C 180,E1 20091.512,E2 20091.512} C_VEL
LIN {X 0,Y 203.056,Z 983.042,A -85,B 0,C 180,E1 20101.463,E2 20101.463} C_VEL
LIN {X 0,Y 215.837,Z 963.961,A -85,B 0,C 180,E1 20110.457,E2 20110.457} C_VEL
LIN {X 0,Y 232.175,Z 938.789,A -85,B 0,C 180,E1 20117.884,E2 20117.884} C_VEL
LIN {X 0,Y 235.517,Z 934.155,A -85,B 0,C 180,E1 20119.058,E2 20119.058} C_VEL
LIN {X 0,Y 244.716,Z 927.511,A -85,B 0,C 180,E1 20121.79,E2 20121.79} C_VEL
LIN {X 0,Y 227.105,Z 934.112,A -85,B 0,C 180,E1 20127.78,E2 20127.78} C_VEL
LIN {X 0,Y 213.274,Z 936.888,A -85,B 0,C 180,E1 20134.8,E2 20134.8} C_VEL
LIN {X 0,Y 203.34,Z 935.57,A -85,B 0,C 180,E1 20142.683,E2 20142.683} C_VEL
LIN {X 0,Y 197.047,Z 928.641,A -85,B 0,C 180,E1 20152.283,E2 20152.283} C_VEL
LIN {X 0,Y 195.341,Z 917.052,A -85,B 0,C 180,E1 20161.12,E2 20161.12} C_VEL
LIN {X 0,Y 195.861,Z 907.128,A -85,B 0,C 180,E1 20166.668,E2 20166.668} C_VEL
LIN {X 0,Y 209.607,Z 898.615,A -85,B 0,C 180,E1 20177.464,E2 20177.464} C_VEL
LIN {X 0,Y 227.279,Z 888.415,A -85,B 0,C 180,E1 20184.602,E2 20184.602} C_VEL
LIN {X 0,Y 241.994,Z 878.893,A -85,B 0,C 180,E1 20188.483,E2 20188.483} C_VEL
LIN {X 0,Y 244.499,Z 877.197,A -85,B 0,C 180,E1 20189.041,E2 20189.041} C_VEL
LIN {X 0,Y 254.916,Z 874.538,A -85,B 0,C 180,E1 20192.511,E2 20192.511} C_VEL
LIN {X 0,Y 255.757,Z 873.95,A -85,B 0,C 180,E1 20192.652,E2 20192.652} C_VEL
LIN {X 0,Y 257.519,Z 872.558,A -85,B 0,C 180,E1 20192.918,E2 20192.918} C_VEL
LIN {X 0,Y 242.052,Z 903.607,A -85,B 0,C 180,E1 20197.475,E2 20197.475} C_VEL
LIN {X 0,Y 225.712,Z 929.68,A -85,B 0,C 180,E1 20203.156,E2 20203.156} C_VEL
LIN {X 0,Y 209.564,Z 952.115,A -85,B 0,C 180,E1 20210.789,E2 20210.789} C_VEL
LIN {X 0,Y 196.707,Z 968.754,A -85,B 0,C 180,E1 20219.98,E2 20219.98} C_VEL
LIN {X 0,Y 189.253,Z 978.816,A -85,B 0,C 180,E1 20228.9,E2 20228.9} C_VEL
LIN {X 0,Y 184.655,Z 985.842,A -85,B 0,C 180,E1 20240.562,E2 20240.562} C_VEL
LIN {X 0,Y 184.042,Z 987.56,A -85,B 0,C 180,E1 20250.001,E2 20250.001} C_VEL
LIN {X 0,Y 184.977,Z 985.316,A -85,B 0,C 180,E1 20260.777,E2 20260.777} C_VEL
LIN {X 0,Y 190.015,Z 977.624,A -85,B 0,C 180,E1 20272.241,E2 20272.241} C_VEL
LIN {X 0,Y 200.151,Z 964.293,A -85,B 0,C 180,E1 20282.796,E2 20282.796} C_VEL
LIN {X 0,Y 213.989,Z 946.126,A -85,B 0,C 180,E1 20291.486,E2 20291.486} C_VEL
LIN {X 0,Y 230.692,Z 921.935,A -85,B 0,C 180,E1 20298.685,E2 20298.685} C_VEL
LIN {X 0,Y 247.06,Z 894.22,A -85,B 0,C 180,E1 20303.966,E2 20303.966} C_VEL
LIN {X 0,Y 258.564,Z 870.051,A -85,B 0,C 180,E1 20307.197,E2 20307.197} C_VEL
LIN {X 0,Y 256.963,Z 850.978,A -85,B 0,C 180,E1 20312.97,E2 20312.97} C_VEL
LIN {X 0,Y 253.451,Z 833.708,A -85,B 0,C 180,E1 20319.611,E2 20319.611} C_VEL
LIN {X 0,Y 249.966,Z 822.103,A -85,B 0,C 180,E1 20325.971,E2 20325.971} C_VEL
LIN {X 0,Y 247.752,Z 815.624,A -85,B 0,C 180,E1 20331.647,E2 20331.647} C_VEL
LIN {X 0,Y 247.252,Z 810.956,A -85,B 0,C 180,E1 20336.482,E2 20336.482} C_VEL
LIN {X 0,Y 247.495,Z 811.764,A -85,B 0,C 180,E1 20343.705,E2 20343.705} C_VEL
LIN {X 0,Y 249.819,Z 818.911,A -85,B 0,C 180,E1 20350.902,E2 20350.902} C_VEL
LIN {X 0,Y 254.427,Z 830.777,A -85,B 0,C 180,E1 20358.106,E2 20358.106} C_VEL
LIN {X 0,Y 259.383,Z 847.203,A -85,B 0,C 180,E1 20364.567,E2 20364.567} C_VEL
LIN {X 0,Y 263.223,Z 866.878,A -85,B 0,C 180,E1 20370.364,E2 20370.364} C_VEL
LIN {X 0,Y 248.57,Z 900.176,A -85,B 0,C 180,E1 20373.908,E2 20373.908} C_VEL
LIN {X 0,Y 232.472,Z 929.052,A -85,B 0,C 180,E1 20378.595,E2 20378.595} C_VEL
LIN {X 0,Y 215.359,Z 955.496,A -85,B 0,C 180,E1 20385.327,E2 20385.327} C_VEL
LIN {X 0,Y 200.095,Z 976.909,A -85,B 0,C 180,E1 20394.095,E2 20394.095} C_VEL
LIN {X 0,Y 189.937,Z 991.875,A -85,B 0,C 180,E1 20403.995,E2 20403.995} C_VEL
LIN {X 0,Y 184.702,Z 1002.19,A -85,B 0,C 180,E1 20415.763,E2 20415.763} C_VEL
LIN {X 0,Y 183.784,Z 1005.972,A -85,B 0,C 180,E1 20425.274,E2 20425.274} C_VEL
LIN {X 0,Y 184.055,Z 1006.519,A -85,B 0,C 180,E1 20429.999,E2 20429.999} C_VEL
LIN {X 0,Y 184.064,Z 1004.552,A -85,B 0,C 180,E1 20439.469,E2 20439.469} C_VEL
LIN {X 0,Y 186.813,Z 997.531,A -85,B 0,C 180,E1 20450.52,E2 20450.52} C_VEL
LIN {X 0,Y 195.141,Z 984.176,A -85,B 0,C 180,E1 20461.751,E2 20461.751} C_VEL
LIN {X 0,Y 207.973,Z 965.995,A -85,B 0,C 180,E1 20470.936,E2 20470.936} C_VEL
LIN {X 0,Y 223.56,Z 943.417,A -85,B 0,C 180,E1 20478.157,E2 20478.157} C_VEL
LIN {X 0,Y 228.016,Z 937.253,A -85,B 0,C 180,E1 20479.785,E2 20479.785} C_VEL
LIN {X 0,Y 233.036,Z 933.996,A -85,B 0,C 180,E1 20481.229,E2 20481.229} C_VEL
LIN {X 0,Y 234.082,Z 932.963,A -85,B 0,C 180,E1 20482.19,E2 20482.19} C_VEL
LIN {X 0,Y 213.112,Z 938.346,A -85,B 0,C 180,E1 20490.189,E2 20490.189} C_VEL
LIN {X 0,Y 200.668,Z 938.436,A -85,B 0,C 180,E1 20497.847,E2 20497.847} C_VEL
LIN {X 0,Y 192.315,Z 934.342,A -85,B 0,C 180,E1 20506.349,E2 20506.349} C_VEL
LIN {X 0,Y 187.874,Z 924.051,A -85,B 0,C 180,E1 20516.545,E2 20516.545} C_VEL
LIN {X 0,Y 187.441,Z 915.885,A -85,B 0,C 180,E1 20522.325,E2 20522.325} C_VEL
LIN {X 0,Y 200.306,Z 907.145,A -85,B 0,C 180,E1 20535.35,E2 20535.35} C_VEL
LIN {X 0,Y 222.513,Z 895.313,A -85,B 0,C 180,E1 20545.177,E2 20545.177} C_VEL
LIN {X 0,Y 240.311,Z 884.559,A -85,B 0,C 180,E1 20549.748,E2 20549.748} C_VEL
LIN {X 0,Y 255.757,Z 873.95,A -85,B 0,C 180,E1 20552.652,E2 20552.652} C_VEL
LIN {X 0,Y 255.733,Z 876.503,A -85,B 0,C 180,E1 20553.386,E2 20553.386} C_VEL
LIN {X 0,Y 252.162,Z 882.848,A -85,B 0,C 180,E1 20553.975,E2 20553.975} C_VEL
LIN {X 0,Y 239.883,Z 899.761,A -85,B 0,C 180,E1 20555.228,E2 20555.228} C_VEL
LIN {X 0,Y 238.457,Z 902.02,A -85,B 0,C 180,E1 20555.584,E2 20555.584} C_VEL
LIN {X 0,Y 221.434,Z 928.52,A -85,B 0,C 180,E1 20561.224,E2 20561.224} C_VEL
LIN {X 0,Y 204.312,Z 951.369,A -85,B 0,C 180,E1 20568.876,E2 20568.876} C_VEL
LIN {X 0,Y 189.835,Z 969.162,A -85,B 0,C 180,E1 20578.774,E2 20578.774} C_VEL
LIN {X 0,Y 180.449,Z 981.07,A -85,B 0,C 180,E1 20590.39,E2 20590.39} C_VEL
LIN {X 0,Y 176.862,Z 986.248,A -85,B 0,C 180,E1 20600.142,E2 20600.142} C_VEL
LIN {X 0,Y 176.175,Z 987.966,A -85,B 0,C 180,E1 20610.001,E2 20610.001} C_VEL
LIN {X 0,Y 177.18,Z 985.726,A -85,B 0,C 180,E1 20621.257,E2 20621.257} C_VEL
LIN {X 0,Y 182.637,Z 978.037,A -85,B 0,C 180,E1 20633.191,E2 20633.191} C_VEL
LIN {X 0,Y 193.478,Z 964.704,A -85,B 0,C 180,E1 20644.079,E2 20644.079} C_VEL
LIN {X 0,Y 207.622,Z 947.099,A -85,B 0,C 180,E1 20652.717,E2 20652.717} C_VEL
LIN {X 0,Y 225.249,Z 922.744,A -85,B 0,C 180,E1 20660.109,E2 20660.109} C_VEL
LIN {X 0,Y 242.219,Z 895.066,A -85,B 0,C 180,E1 20665.416,E2 20665.416} C_VEL
LIN {X 0,Y 252.997,Z 873.977,A -85,B 0,C 180,E1 20668.227,E2 20668.227} C_VEL
LIN {X 0,Y 252.271,Z 856.274,A -85,B 0,C 180,E1 20673.76,E2 20673.76} C_VEL
LIN {X 0,Y 249.486,Z 839.481,A -85,B 0,C 180,E1 20680.494,E2 20680.494} C_VEL
LIN {X 0,Y 246.633,Z 828.397,A -85,B 0,C 180,E1 20686.996,E2 20686.996} C_VEL
LIN {X 0,Y 244.852,Z 818.843,A -85,B 0,C 180,E1 20696.447,E2 20696.447} C_VEL
LIN {X 0,Y 244.852,Z 818.19,A -85,B 0,C 180,E1 20699.992,E2 20699.992} C_VEL
LIN {X 0,Y 245.193,Z 820.582,A -85,B 0,C 180,E1 20704.716,E2 20704.716} C_VEL
LIN {X 0,Y 247.048,Z 826.208,A -85,B 0,C 180,E1 20710.586,E2 20710.586} C_VEL
LIN {X 0,Y 250.933,Z 837.421,A -85,B 0,C 180,E1 20717.55,E2 20717.55} C_VEL
LIN {X 0,Y 255.151,Z 853.574,A -85,B 0,C 180,E1 20724.068,E2 20724.068} C_VEL
LIN {X 0,Y 257.832,Z 870.068,A -85,B 0,C 180,E1 20729.16,E2 20729.16} C_VEL
LIN {X 0,Y 242.861,Z 902.308,A -85,B 0,C 180,E1 20732.685,E2 20732.685} C_VEL
LIN {X 0,Y 225.102,Z 932.48,A -85,B 0,C 180,E1 20737.782,E2 20737.782} C_VEL
LIN {X 0,Y 207.634,Z 957.775,A -85,B 0,C 180,E1 20744.684,E2 20744.684} C_VEL
LIN {X 0,Y 192.099,Z 978.482,A -85,B 0,C 180,E1 20753.761,E2 20753.761} C_VEL
LIN {X 0,Y 181.839,Z 992.824,A -85,B 0,C 180,E1 20764.077,E2 20764.077} C_VEL
LIN {X 0,Y 176.913,Z 1001.776,A -85,B 0,C 180,E1 20775.122,E2 20775.122} C_VEL
LIN {X 0,Y 175.889,Z 1005.563,A -85,B 0,C 180,E1 20785.061,E2 20785.061} C_VEL
LIN {X 0,Y 176.177,Z 1006.113,A -85,B 0,C 180,E1 20789.999,E2 20789.999} C_VEL
LIN {X 0,Y 176.18,Z 1004.141,A -85,B 0,C 180,E1 20799.896,E2 20799.896} C_VEL
